Yaskawa INFORM job: OK_R2_O57-69(1)(90,0)OLDMAREK.JBI

/JOB
//NAME OK_R2_O57-69(1)(90,0)OLDMAREK
//POS
///NPOS 679,679,679,19,0,0
///TOOL 0
///POSTYPE PULSE
///PULSE
C00000=-115282,71817,32941,48127,54711,-22306
C00001=-113844,78377,40832,48113,52960,-22533
C00002=-113286,81152,44222,48167,52223,-22657
C00003=-112658,81907,45149,47913,51773,-22558
C00004=-113286,81152,44222,48167,52223,-22657
C00005=-114841,82290,45172,49039,53033,-23084
C00006=-115003,85006,48527,49507,52672,-23414
C00007=-114841,82290,45172,49039,53033,-23084
C00008=-115410,79539,41800,48987,53774,-22957
C00009=-116878,73048,33960,49005,55537,-22725
C00010=-112638,83822,30523,28584,74380,-13794
C00011=-107672,118155,51647,4031,94928,-4029
C00012=-107420,122850,61171,3935,91477,-4062
C00013=-107323,125066,65433,3902,89992,-4078
C00014=-107323,124239,65578,3901,89479,-4094
C00015=-107323,125066,65433,3902,89992,-4078
C00016=-107335,126122,66498,3905,89879,-4086
C00017=-107232,129619,71327,3873,88703,-4090
C00018=-107335,126122,66498,3905,89879,-4086
C00019=-107432,123868,62180,3938,91380,-4069
C00020=-107683,119107,52557,4034,94858,-4034
C00021=-108242,110727,51927,9928,92581,-10453
C00022=-107623,115488,61342,9730,89211,-10523
C00023=-107381,117723,65553,9663,87760,-10558
C00024=-107381,117129,66014,9664,87180,-10602
C00025=-107381,117723,65553,9663,87760,-10558
C00026=-107320,118492,66386,9646,87637,-10548
C00027=-107068,121743,70795,9581,86581,-10547
C00028=-107320,118492,66386,9646,87637,-10548
C00029=-107562,116223,62127,9713,89100,-10512
C00030=-108179,111405,52627,9909,92492,-10440
C00031=-110424,91387,35110,11931,86832,-11135
C00032=-122323,33946,36249,27998,48832,-19209
C00033=-121111,41698,46132,28269,46563,-19325
C00034=-120645,45031,50436,28448,45578,-19411
C00035=-120645,45990,52788,28899,44735,-19701
C00036=-120645,45031,50436,28448,45578,-19411
C00037=-120832,44203,49576,28499,45733,-19457
C00038=-120451,46607,52174,28466,45283,-19410
C00039=-120832,44203,49576,28499,45733,-19457
C00040=-121303,40901,45320,28328,46708,-19376
C00041=-122523,33209,35531,28074,48955,-19270
C00042=-138494,21467,-20962,-13510,88545,-918
C00043=-172308,65494,48979,-45567,35920,22282
C00044=-172307,66906,54819,-48573,33928,23926
C00045=-172639,69838,58273,-49022,33332,24169
C00046=-173239,69159,57471,-48394,33104,23833
C00047=-173424,69192,57512,-48260,33005,23761
C00048=-172268,71224,59921,-49648,33330,24503
C00049=-172150,82507,73646,-52983,31698,26274
C00050=-172069,85080,76852,-53896,31347,26756
C00051=-171567,71541,60313,-50254,33662,24828
C00052=-171245,62238,49417,-48357,35120,23797
C00053=-171365,58220,44512,-47276,35710,23205
C00054=-172568,85923,51709,-38156,42478,18009
C00055=-173210,88622,55081,-38109,41654,18042
C00056=-173399,87523,53708,-37764,41797,17852
C00057=-171913,88923,55458,-39192,42161,18576
C00058=-172373,102262,72497,-41555,39146,20013
C00059=-172364,103826,74533,-41931,38810,20229
C00060=-172120,93439,61160,-39872,41141,19005
C00061=-171772,85324,50969,-38678,42942,18248
C00062=-171214,82198,47055,-38587,43820,18132
C00063=-172412,95660,50695,-34930,47113,15937
C00064=-172941,98291,54078,-34907,46302,16003
C00065=-173393,98042,53756,-34511,46183,15812
C00066=-173582,97646,53244,-34301,46202,15703
C00067=-172217,98411,54230,-35491,46558,16277
C00068=-172267,109740,69033,-37375,43863,17490
C00069=-172235,113172,73586,-38066,43046,17916
C00070=-172202,103053,60251,-36243,45483,16763
C00071=-171971,91033,44794,-34631,48320,15659
C00072=-172583,89506,42865,-33959,48423,15307
C00073=-136545,44574,15947,-43124,46451,20365
C00074=-172050,-124043,-93312,-19428,16171,9287
C00075=-153076,-24082,-53998,12354,68401,18517
C00076=-141616,-19382,-55807,13562,72328,27791
C00077=-136367,-32764,-63918,14399,72043,28923
C00078=-134539,-35777,-64067,14758,71094,29221
C00079=-134539,-36232,-63095,14829,70289,29119
C00080=-134539,-35777,-64067,14758,71094,29221
C00081=-134790,5262,-45049,12672,103577,12599
C00082=-134622,7343,-43237,12633,103510,12643
C00083=-134790,5262,-45049,12672,103577,12599
C00084=-132608,-4947,-51631,7718,96928,11812
C00085=-133594,-4601,-51352,7990,97018,11521
C00086=-132608,-4947,-51631,7718,96928,11812
C00087=-132561,-6063,-53863,7723,97717,11875
C00088=-132436,-8720,-59337,7740,99694,12036
C00089=-132445,-1782,-62924,7952,105415,12403
C00090=-141601,37323,-23290,10329,102010,9516
C00091=-93172,55874,9388,-1843,94357,23900
C00092=-93485,56784,11787,-1769,93341,23816
C00093=-93485,56329,12545,-1767,92641,23826
C00094=-93485,56784,11787,-1769,93341,23816
C00095=-93464,57012,11403,-1775,93695,23818
C00096=-93714,59095,13766,-1718,93307,23745
C00097=-93464,57012,11403,-1775,93695,23818
C00098=-94351,55649,10247,-1575,93690,23540
C00099=-95033,54913,9421,-1421,93808,23324
C00100=-94351,55649,10247,-1575,93690,23540
C00101=-94041,54751,7862,-1648,94701,23624
C00102=-93250,52756,2164,-1838,97197,23834
C00103=-93258,57323,-1415,-1867,101744,23764
C00104=-108708,74058,35602,41753,92549,11625
C00105=-107609,77867,43172,41468,89995,11080
C00106=-107179,79572,46434,41382,88936,10847
C00107=-107179,79487,47575,41378,88368,10623
C00108=-107179,79572,46434,41382,88936,10847
C00109=-85041,17756,-8276,-11251,50625,9461
C00110=-85416,19690,-6470,-10982,50459,9320
C00111=-85041,17756,-8276,-11251,50625,9461
C00112=-87036,75660,30192,-3211,91902,25887
C00113=-87645,74633,28952,-3076,92115,25688
C00114=-87036,75660,30192,-3211,91902,25887
C00115=-86708,74680,27642,-3289,92979,25963
C00116=-85872,72543,21626,-3493,95611,26155
C00117=-85876,74587,19798,-3512,97782,26092
C00118=-86821,26768,-33196,-3418,105774,25582
C00119=-56288,-65443,-100505,-9939,102051,34984
C00120=-94872,-76247,-37251,-15619,10327,-42827
C00121=-113351,-68967,-59155,816,27582,-73246
C00122=-112415,-66495,-57032,-529,27544,-72574
C00123=-112416,-66088,-55565,-540,26850,-72568
C00124=-112415,-66495,-57032,-529,27544,-72574
C00125=-125986,-60936,-52893,34026,33366,-67517
C00126=-125619,-58716,-51713,33325,33568,-67144
C00127=-125986,-60936,-52893,34026,33366,-67517
C00128=-125164,-63316,-53721,33839,32440,-67422
C00129=-123797,-63897,-54019,32563,31806,-66752
C00130=-125164,-63316,-53721,33839,32440,-67422
C00131=-126284,-65474,-55722,34821,32994,-67941
C00132=-120687,-90156,-48971,65843,10407,33929
C00133=-163424,-29173,-12092,69684,68620,47205
C00134=-154639,-8126,3338,68913,63218,49031
C00135=-170775,-70491,-60275,67726,76450,43734
C00136=-168988,-72616,-61292,67687,75067,43782
C00137=-168256,-73449,-61686,67672,74502,43804
C00138=-168255,-73444,-61683,67672,74502,43805
C00139=-168256,-73449,-61686,67672,74502,43804
C00140=-168129,-73592,-61753,67670,74405,43808
C00141=-167340,-74469,-62163,67655,73798,43833
C00142=-168129,-73592,-61753,67670,74405,43808
C00143=-168863,-72760,-61361,67684,74971,43786
C00144=-170655,-70639,-60347,67723,76357,43737
C00145=-172135,-82938,-72310,60788,72518,32969
C00146=-200540,-66438,-67217,63628,100285,-15829
C00147=-127293,-88890,-117674,21964,112183,-47373
C00148=-127884,-113870,-117586,20406,100261,-49782
C00149=-127000,-93154,-82052,19489,96345,-50169
C00150=-123343,-94047,-79271,19637,93420,-49322
C00151=-121848,-94244,-78089,19702,92278,-48969
C00152=-121841,-92834,-76346,19694,91947,-49020
C00153=-121848,-94244,-78089,19702,92278,-48969
C00154=-119969,-93354,-78147,19815,92288,-48290
C00155=-118222,-93288,-78121,19899,91881,-47727
C00156=-119969,-93354,-78147,19815,92288,-48290
C00157=-121462,-93189,-79339,19761,93422,-48643
C00158=-125120,-92380,-82146,19635,96326,-49491
C00159=-116413,-89407,-85315,-11170,94586,69972
C00160=-118284,-91858,-82643,-11111,91478,69605
C00161=-119058,-92674,-81496,-11095,90266,69446
C00162=-119072,-91347,-79783,-11093,89899,69474
C00163=-119058,-92674,-81496,-11095,90266,69446
C00164=-118796,-98042,-83265,-11090,88662,69679
C00165=-118746,-100551,-83769,-11090,87708,69781
C00166=-118796,-98042,-83265,-11090,88662,69679
C00167=-123354,-93602,-81963,-11047,89491,68033
C00168=-125085,-93483,-81915,-11019,89286,67454
C00169=-123354,-93602,-81963,-11047,89491,68033
C00170=-122534,-92869,-83147,-11066,90689,68210
C00171=-120547,-90622,-85912,-11132,93767,68620
C00172=-120571,-90661,-98380,-11386,101275,67925
C00173=-125069,-105236,-119201,46912,96955,7142
C00174=-121279,-99548,-114464,46207,95099,8000
C00175=-119841,-97303,-112552,45921,94382,8319
C00176=-119849,-96483,-111054,45883,94032,8153
C00177=-119841,-97303,-112552,45921,94382,8319
C00178=-121259,-87971,-110760,46601,97668,9229
C00179=-121544,-83907,-109504,46842,98723,9610
C00180=-121259,-87971,-110760,46601,97668,9229
C00181=-122654,-89805,-112582,46929,98462,8982
C00182=-126320,-94321,-117059,47765,100534,8329
C00183=-125132,-111985,-108710,18887,62200,-22139
C00184=-122150,-102499,-103347,17190,63051,-20837
C00185=-121052,-98905,-101202,16573,63333,-20372
C00186=-121051,-97751,-99591,16628,62949,-20429
C00187=-121052,-98905,-101202,16573,63333,-20372
C00188=-120662,-97381,-100799,16308,63770,-20159
C00189=-118912,-97325,-100778,15434,63451,-19540
C00190=-120662,-97381,-100799,16308,63770,-20159
C00191=-120717,-96579,-100674,16290,64103,-20131
C00192=-120723,-93199,-99767,16143,65237,-19969
C00193=-120717,-96579,-100674,16290,64103,-20131
C00194=-121791,-100117,-102825,16885,63842,-20577
C00195=-124704,-109452,-108202,18522,63043,-21827
C00196=-114740,-109793,-107699,-22238,66313,27441
C00197=-118303,-101714,-102676,-20552,66389,26052
C00198=-119630,-98598,-100655,-19919,66404,25543
C00199=-119640,-97443,-99041,-19972,66025,25607
C00200=-119630,-98598,-100655,-19919,66404,25543
C00201=-120869,-98346,-100801,-19339,66320,25087
C00202=-122629,-98310,-100787,-18548,65929,24486
C00203=-120869,-98346,-100801,-19339,66320,25087
C00204=-120753,-95574,-99975,-19267,67213,24978
C00205=-120759,-92226,-99069,-19116,68313,24791
C00206=-120753,-95574,-99975,-19267,67213,24978
C00207=-119475,-98647,-102011,-19875,67204,25461
C00208=-116042,-106621,-107071,-21497,67130,26779
C00209=-113894,-113482,-108593,-25442,60982,30098
C00210=-117729,-104898,-103745,-23262,61171,28471
C00211=-119152,-101582,-101788,-22448,61245,27877
C00212=-119170,-99953,-99618,-22541,60778,27968
C00213=-119152,-101582,-101788,-22448,61245,27877
C00214=-121013,-102333,-103012,-21430,61098,27156
C00215=-123420,-102254,-102982,-20177,60519,26301
C00216=-121013,-102333,-103012,-21430,61098,27156
C00217=-120862,-89775,-98642,-20835,64658,26523
C00218=-120866,-85351,-97357,-20602,66047,26262
C00219=-120862,-89775,-98642,-20835,64658,26523
C00220=-119577,-92842,-100627,-21537,64647,27018
C00221=-116128,-100765,-105545,-23412,64594,28369
C00222=-120616,-96668,-103675,-23957,64374,45643
C00223=-120616,-97077,-101536,-24254,62975,45956
C00224=-120616,-97187,-100661,-24377,62430,46080
C00225=-118869,-97129,-100639,-25236,62958,46664
C00226=-120614,-98300,-102259,-24293,62807,45995
C00227=-120617,-94441,-109322,-23464,92098,42048
C00228=-120616,-97113,-101199,-23421,86229,43199
C00229=-120616,-97196,-100378,-23430,85724,43299
C00230=-120616,-97068,-101477,-23418,86408,43164
C00231=-120616,-96536,-104145,-23405,88172,42819
C00232=-120615,-97089,-97846,-24331,46439,48575
C00233=-120614,-96205,-89198,-26458,42021,49913
C00234=-120613,-95813,-87227,-26966,41113,50220
C00235=-120613,-95637,-86431,-27175,40755,50344
C00236=-118868,-95589,-86413,-28580,41350,51125
C00237=-120611,-96965,-88121,-26990,41076,50233
C00238=-120617,-95981,-105264,-23408,89069,42643
C00239=-120616,-96766,-101896,-23413,86788,43090
C00240=-120616,-96795,-102141,-18817,118956,36582
C00241=-120616,-96568,-103294,-18987,119739,36439
C00242=-120617,-95735,-106079,-19458,121767,36056
C00243=-120683,-72727,-118704,-1403,106780,1205
C00244=-120616,-97110,-101484,23732,56591,-46685
C00245=-120615,-97329,-97421,24453,54195,-47265
C00246=-120615,-97216,-95276,24833,53043,-47558
C00247=-120615,-97137,-94405,24989,52592,-47675
C00248=-120613,-98372,-96050,24869,52935,-47585
C00249=-122362,-97116,-94396,26052,53130,-48332
C00250=-120617,-95602,-107135,23341,90098,-42167
C00251=-120617,-96025,-106062,23332,89289,-42325
C00252=-120617,-96280,-105304,23328,88738,-42432
C00253=-120617,-95942,-106325,23333,89477,-42288
C00254=-120617,-94838,-108784,23367,91395,-41914
C00255=-120619,-89077,-114974,23678,97628,-40680
C00256=-119375,-87803,-114046,-9627,73434,-76892
C00257=-119874,-91001,-111320,-9540,70103,-76790
C00258=-120074,-92022,-110137,-9508,68845,-76756
C00259=-120388,-88035,-108953,-9268,70114,-76963
C00260=-120068,-92699,-111595,-9479,69387,-76797
C00261=-120617,-92323,-109789,-9348,67950,-76861
C00262=-120617,-92636,-109412,-9435,67087,-76774
C00263=-120617,-92966,-108935,-9385,65680,-76698
C00264=-120617,-93485,-108112,-8702,63167,-76584
C00265=-120617,-93807,-107566,-7310,61334,-76551
C00266=-120617,-93899,-107425,-5913,60596,-76588
C00267=-120617,-91887,-110532,-5160,63404,-76609
C00268=-120617,-91830,-110616,-4244,63440,-76636
C00269=-120617,-91600,-110911,-2665,64017,-76695
C00270=-120618,-91126,-111456,-1065,65432,-76762
C00271=-120618,-90436,-112164,126,67515,-76814
C00272=-120618,-89799,-112749,669,69377,-76843
C00273=-120618,-88579,-113586,734,71430,-76721
C00274=-120618,-87737,-114188,674,73665,-76767
C00275=-120618,-86710,-114840,-40,76341,-76871
C00276=-120619,-85981,-115253,-1370,78289,-77032
C00277=-120619,-85769,-115356,-2649,79041,-77176
C00278=-118258,-89310,-112812,-4565,75923,-76275
C00279=-117029,-89279,-112689,-5985,75998,-75947
C00280=-115084,-89307,-112300,-8369,75681,-75412
C00281=-113300,-89514,-111627,-10775,74614,-74872
C00282=-112191,-89952,-110802,-12600,72842,-74453
C00283=-112162,-90329,-110382,-13115,71673,-74372
C00284=-116808,-91534,-110372,-11031,70029,-75758
C00285=-120074,-92022,-110137,-9508,68845,-76756
C00286=-119874,-91001,-111320,-9540,70103,-76790
C00287=-119375,-87803,-114046,-9627,73434,-76892
C00288=-120613,-96141,-86612,-20456,81391,53018
C00289=-120613,-95201,-83022,-20541,79769,53295
C00290=-120613,-94772,-81561,-20579,79132,53405
C00291=-119108,-93506,-81277,-20755,79958,53812
C00292=-120703,-96226,-83293,-20548,79408,53324
C00293=-120613,-95341,-83418,-16256,85806,57019
C00294=-120612,-93770,-78536,-16295,83694,57299
C00295=-120612,-93943,-79000,-13291,89893,68155
C00296=-120613,-94474,-80645,-13297,90613,68078
C00297=-120613,-95649,-84682,-13324,92446,67881
C00298=-120615,-97441,-93706,-13451,96957,67391
C00299=-117944,-114132,-91182,23549,57658,-33742
C00300=-120612,-94052,-79174,30375,49115,-27391
C00301=-120612,-92306,-74262,31338,47277,-28046
C00302=-120611,-91624,-72518,31687,46656,-28277
C00303=-120611,-91343,-71816,31829,46409,-28371
C00304=-120609,-92783,-73582,31657,46706,-28257
C00305=-122365,-91326,-71808,32798,47083,-29054
C00306=-120614,-96423,-87542,23693,78601,-44429
C00307=-120612,-92192,-73989,24270,72943,-45595
C00308=-120612,-92493,-74805,23528,86971,-60762
C00309=-120612,-93040,-76284,23523,87550,-60648
C00310=-120612,-94304,-79928,23524,89017,-60360
C00311=-192979,-49879,-84133,31949,90821,-59300
C00312=-226136,-49296,-77583,43048,96139,-60221
C00313=-194231,-43574,-37464,64429,96533,35524
C00314=-168190,-921,2356,69742,86936,65420
C00315=-157686,-14873,-8721,69811,79682,66593
C00316=-155170,-17431,-10634,69793,77924,66853
C00317=-154140,-18406,-11354,69782,77205,66960
C00318=-154960,-19735,-12328,69815,77730,66818
C00319=-154139,-18877,-12975,69638,77486,67291
C00320=-152416,-19959,-12491,68149,70274,62953
C00321=-151462,-20771,-13080,67326,65877,57651
C00322=-150584,-21490,-13598,66880,61935,51327
C00323=-149448,-22378,-14235,66195,57985,45258
C00324=-150364,-21665,-13724,66599,59939,44567
C00325=-146294,-24621,-15825,64622,49633,44461
C00326=-147024,-24129,-15478,65026,50858,44122
C00327=-148183,-23314,-14902,65711,53127,43519
C00328=-150746,-21357,-13503,66515,56405,42739
C00329=-151844,-20450,-12847,67017,58691,42205
C00330=-154160,-18394,-11345,67568,61790,41547
C00331=-155150,-17454,-10651,67918,63984,41080
C00332=-156307,-16307,-9798,68285,66690,40524
C00333=-158578,-13896,-7981,68632,70174,39857
C00334=-158236,-14274,-8267,68563,69306,40027
C00335=-158768,-13688,-7823,68593,69674,39964
C00336=-160083,-12191,-6676,68663,70584,39811
C00337=-163356,-38025,-17867,70039,68206,46757
C00338=-171321,-47804,-23743,70196,73038,45095
C00339=-120855,-117042,-83065,287,50429,-281
C00340=-120852,-56541,-79529,233,79340,-219
C00341=-120696,51333,26745,175,69370,-180
C00342=-120686,107948,75662,172,68359,-178
C00343=-120686,108277,78684,174,66668,-180
C00344=-120686,108491,80003,175,65967,-181
C00345=-120685,108330,78544,174,66782,-180
C00346=-120704,104314,74519,181,67195,-186
C00347=-120686,108513,80202,3786,65964,-3429
C00348=-120686,108564,80691,8354,65806,-7433
C00349=-120686,108545,80707,11489,66690,-7514
C00350=-120686,108555,80692,12508,67155,-8479
C00351=-120686,108564,80762,15450,68398,-11287
C00352=-120686,108549,80793,17539,69495,-16102
C00353=-120686,109188,83963,29512,74271,-26746
C00354=-120686,108838,82574,29428,74862,-26590
C00355=-120686,108172,79385,29242,76284,-26220
C00356=-120686,107962,76375,6322,66410,-5366
C00357=-120686,108346,79348,6400,64788,-5455
C00358=-120686,108578,80641,6435,64115,-5493
C00359=-120686,108293,79018,6392,64962,-5445
C00360=-120992,104893,75799,6510,65219,-5544
C00361=-120686,108263,79465,19749,71998,-15740
C00362=-120686,108289,79502,19750,71989,-15741
C00363=-120686,109192,84126,33583,78410,-30786
C00364=-120686,108845,82779,33520,78957,-30620
C00365=-120686,108177,79678,33383,80274,-30223
C00366=-146832,94827,54018,-31343,96631,42054
C00367=-156862,88199,54516,-55770,96758,71489
C00368=-156858,88352,61458,-55305,94312,73083
C00369=-157852,91445,67330,-55099,92539,73648
C00370=-158245,92835,69884,-55033,91801,73892
C00371=-157951,96204,74186,-54996,91433,74294
C00372=-157784,91273,67188,-55102,92578,73662
C00373=-158040,92399,69988,-55026,91755,74041
C00374=-159291,95627,71523,-51291,93332,81554
C00375=-160209,98279,73182,-48482,94322,83905
C00376=-159956,97162,70645,-48575,95125,83623
C00377=-159321,94794,64867,-48849,97041,82959
C00378=-174197,80542,71118,-15802,102714,62389
C00379=-174195,80556,71135,-15802,102711,62390
C00380=-174195,80561,71142,-15801,102710,62390
C00381=-173773,83477,74756,-15654,102092,62625
C00382=-174194,79765,68888,-15876,103653,62265
C00383=-174199,80535,71109,-11568,105990,64366
C00384=-174198,80539,71114,-12074,105866,67869
C00385=-174201,80518,71089,-8660,108894,72599
C00386=-174202,80510,71078,-8661,108896,72599
C00387=-174205,80488,71052,-8662,108901,72597
C00388=-174210,80448,71002,-8664,108910,72595
C00389=-160796,99181,68474,-21491,79626,-54117
C00390=-160795,99200,68498,-21491,79622,-54116
C00391=-160795,99207,68507,-21491,79620,-54116
C00392=-160747,98987,66984,-21457,80402,-54239
C00393=-161332,101028,70752,-21395,79065,-54211
C00394=-160795,99207,68507,-21491,79620,-54116
C00395=-160795,99200,68498,-21491,79622,-54116
C00396=-160796,99181,68474,-21491,79626,-54117
C00397=-156887,88424,61529,-55303,94292,73080
C00398=-157880,91522,67408,-55097,92517,73646
C00399=-158273,92915,69967,-55032,91779,73890
C00400=-157979,96289,74274,-54994,91410,74293
C00401=-157812,91350,67266,-55100,92556,73660
C00402=-158068,92478,70069,-55024,91733,74039
C00403=-159318,95712,71612,-51289,93309,81552
C00404=-160236,98368,73278,-48480,94299,83903
C00405=-159983,97249,70737,-48574,95102,83621
C00406=-159349,94875,64951,-48847,97020,82956
C00407=-174197,80542,71118,-15802,102714,62389
C00408=-174195,80555,71135,-15802,102711,62390
C00409=-174195,80561,71141,-15801,102710,62390
C00410=-173773,83477,74755,-15654,102093,62624
C00411=-174194,79764,68887,-15876,103653,62265
C00412=-174199,80534,71109,-11568,105990,64366
C00413=-174198,80538,71114,-12074,105866,67869
C00414=-174201,80518,71088,-8660,108894,72599
C00415=-174202,80509,71078,-8661,108896,72599
C00416=-174205,80488,71051,-8662,108901,72597
C00417=-174210,80448,71002,-8664,108910,72595
C00418=-160796,99181,68473,-21491,79626,-54117
C00419=-160795,99199,68497,-21491,79622,-54116
C00420=-160795,99206,68506,-21491,79620,-54116
C00421=-160747,98986,66983,-21457,80402,-54239
C00422=-161332,101028,70752,-21395,79065,-54211
C00423=-160795,99206,68506,-21491,79620,-54116
C00424=-160795,99199,68497,-21491,79622,-54116
C00425=-160796,99181,68473,-21491,79626,-54117
C00426=-156915,88496,61599,-55301,94271,73077
C00427=-157907,91600,67487,-55096,92496,73644
C00428=-158301,92995,70050,-55030,91757,73888
C00429=-158006,96373,74363,-54993,91387,74291
C00430=-157840,91427,67345,-55098,92535,73658
C00431=-158096,92558,70151,-55023,91711,74037
C00432=-159346,95797,71702,-51288,93287,81550
C00433=-160263,98458,73375,-48479,94275,83902
C00434=-160010,97336,70829,-48572,95080,83619
C00435=-159376,94956,65035,-48845,96998,82954
C00436=-174177,99010,68236,-17004,113547,60859
C00437=-174175,99024,68253,-17003,113544,60860
C00438=-174175,99029,68260,-17002,113542,60860
C00439=-173779,101892,71964,-16797,112849,61119
C00440=-174174,98966,66934,-17118,114293,60744
C00441=-174178,99003,68226,-12626,117020,63205
C00442=-174178,99007,68232,-13170,116875,66659
C00443=-174181,98987,68205,-9575,120026,71701
C00444=-174182,98978,68194,-9576,120028,71701
C00445=-174185,98957,68167,-9578,120033,71699
C00446=-174189,98918,68117,-9580,120044,71697
C00447=-160796,99180,68472,-21491,79627,-54117
C00448=-160795,99198,68496,-21491,79622,-54116
C00449=-160795,99206,68506,-21491,79620,-54116
C00450=-160747,98986,66982,-21457,80402,-54239
C00451=-161332,101027,70751,-21395,79065,-54211
C00452=-160795,99206,68506,-21491,79620,-54116
C00453=-160795,99198,68496,-21491,79622,-54116
C00454=-160796,99180,68472,-21491,79627,-54117
C00455=-160394,63694,17038,-3651,83782,-73608
C00456=-190015,-23229,-64935,6709,90053,81130
C00457=-200263,9721,-38620,10181,91724,78169
C00458=-174135,-51322,-31088,61328,33879,50976
C00459=-174134,-51319,-31087,61327,33879,50977
C00460=-174133,-51978,-32760,60430,34229,51462
C00461=-175008,-52913,-31974,62066,34294,50529
C00462=-174165,-51376,-31119,68078,48326,49661
C00463=-174167,-51380,-31120,67173,48568,55955
C00464=-174192,-51426,-31146,69828,61157,64510
C00465=-174196,-51432,-31150,69829,61158,64509
C00466=-160788,-42263,-32458,15580,47921,8219
C00467=-160788,-42263,-32458,15580,47921,8219
C00468=-159909,-43388,-33874,14966,48039,8647
C00469=-161405,-44119,-33586,16024,47791,7908
C00470=-160787,-42259,-32456,15583,47920,8217
C00471=-160784,-42250,-32450,15581,47921,8219
C00472=-160783,-42246,-32448,15576,47922,8221
C00473=-160783,-42246,-32448,15576,47922,8221
C00474=-146637,-39575,-34461,6046,48590,14746
C00475=-174196,-30579,-7118,69980,41906,48750
C00476=-174191,-30568,-7111,69979,41904,48752
C00477=-174188,-30559,-7105,69977,41901,48753
C00478=-174186,-30555,-7102,69976,41901,48754
C00479=-174186,-31355,-8970,69207,42176,49221
C00480=-174962,-32094,-8117,70258,42357,48510
C00481=-174194,-30569,-7112,71825,47591,46341
C00482=-174196,-30575,-7115,70727,48120,54586
C00483=-174217,-30615,-7142,71977,59732,62495
C00484=-174219,-30621,-7146,71977,59734,62495
C00485=-174226,-30637,-7157,71978,59738,62493
C00486=-174235,-30659,-7171,71979,59742,62491
C00487=-160826,40415,13631,53464,67015,37205
C00488=-160826,40346,14725,53699,66583,36924
C00489=-160826,40419,13556,53448,67045,37224
C00490=-161205,38368,12671,53745,66948,36941
C00491=-160829,40326,14814,56358,71294,34357
C00492=-160833,40301,19018,62693,68392,39666
C00493=-160845,41308,28286,76228,74003,43895
C00494=-160845,41098,27088,76066,74172,44186
C00495=-160847,40669,24199,75673,74598,44902
C00496=-160844,40222,15431,74465,76073,47261
C00497=-107800,-52207,-58944,57218,40703,55200
C00498=-68476,-97884,-84022,-50002,23247,45036
C00499=-66040,-99229,-83751,-49838,32871,-40371
C00500=-120096,-126434,-88762,51835,16555,74218
C00501=-135002,-84086,-73993,57476,43061,70498
C00502=-132040,-84680,-73570,56549,40955,71010
C00503=-130846,-84617,-72526,56532,39890,71007
C00504=-131406,-87072,-73560,57444,39877,70476
C00505=-130845,-85029,-73961,55869,40275,71397
C00506=-120674,-85352,-72158,6203,19725,75700
C00507=-120674,-85360,-72169,6198,19735,75701
C00508=-120674,-85375,-72170,13051,20123,72466
C00509=-120675,-85403,-72185,17568,20556,70326
C00510=-120675,-85415,-72191,21840,21109,68297
C00511=-120675,-85426,-72197,23876,21425,67327
C00512=-120675,-85665,-72942,26166,23375,58358
C00513=-120894,-85673,-72945,29533,24131,56524
C00514=-120675,-85602,-72710,24864,23359,52833
C00515=-120675,-85601,-72708,24818,23350,52837
C00516=-120675,-85948,-73873,24306,23842,53086
C00517=-120674,-86249,-74914,23862,24287,53303
C00518=-120096,-126434,-88762,51835,16555,74218
C00519=-66040,-99229,-83751,-49838,32871,-40371
C00520=-124550,-62434,-86348,-29573,82344,852
C00521=-123235,4833,-40404,-29868,88268,-211
C00522=-160797,40338,30634,-17216,54639,-7315
C00523=-160798,40335,30631,-17216,54639,-7316
C00524=-160798,40334,30630,-17216,54639,-7316
C00525=-160254,39145,28669,-17377,55324,-7200
C00526=-161179,38217,28428,-16962,54815,-7509
C00527=-160797,40338,30635,-17214,54636,-7317
C00528=-160796,40349,30645,-17215,54635,-7316
C00529=-160795,40353,30650,-17218,54637,-7314
C00530=-160795,40355,30652,-17218,54637,-7314
C00531=-160794,40358,30655,-17219,54637,-7314
C00532=-134055,6389,-12297,-27269,70214,305
C00533=-134055,6386,-12300,-27269,70214,304
C00534=-134056,6385,-12301,-27269,70214,304
C00535=-133336,6111,-13253,-27465,70843,431
C00536=-134209,4258,-14137,-27207,70198,248
C00537=-134055,6389,-12297,-27268,70211,304
C00538=-134055,6399,-12288,-27268,70211,304
C00539=-134055,6404,-12285,-27269,70214,305
C00540=-134054,6405,-12283,-27269,70214,305
C00541=-134054,6409,-12280,-27270,70214,305
C00542=-134054,6381,-12304,-27269,70214,305
C00543=-107307,118486,66692,6711,86217,-7198
C00544=-107308,118513,66728,6711,86209,-7198
C00545=-107308,118524,66743,6711,86205,-7199
C00546=-107412,115203,62263,6738,87257,-7176
C00547=-107308,119140,66313,6709,86782,-7168
C00548=-107310,118572,66809,-801,85169,-3247
C00549=-107308,118507,66720,-802,85190,-3246
C00550=-107307,118486,66692,-801,85189,-3246
C00551=-107307,118478,66681,-801,85191,-3246
C00552=-107306,118457,66653,-801,85198,-3245
C00553=-107310,127854,66507,14056,94097,-10874
C00554=-107310,125830,66726,14028,92956,-11004
C00555=-107310,125066,66876,14018,92485,-11057
C00556=-107310,125885,66724,14029,92985,-11000
C00557=-107565,122036,62719,14104,93498,-11023
C00558=-107311,125084,66901,14017,92482,-11058
C00559=-107312,125131,66974,14017,92463,-11061
C00560=-107313,125147,66999,14019,92452,-11062
C00561=-107313,125910,66849,14028,92923,-11008
C00562=-107313,127932,66629,14055,94064,-10878
C00563=-132655,20555,-34602,20500,105579,-17250
C00564=-120395,-75677,-109491,17431,99945,-14261
C00565=-120731,-81008,-115648,-105,86416,-81801
C00566=-120675,-24649,-47159,-132,73228,-81771
C00567=-120676,-24635,-47149,-131,73230,-81771
C00568=-120677,-24629,-47145,-131,73230,-81771
C00569=-120676,-24365,-48211,-131,74022,-81772
C00570=-121750,-24621,-47139,317,73232,-82133
C00571=-120677,-24629,-47145,-131,73230,-81771
C00572=-120676,-24635,-47149,-131,73230,-81771
C00573=-120675,-24649,-47159,-132,73228,-81771
C00574=-86683,-40445,-63075,-13763,77736,-70672
C00575=-103499,26970,-9106,-7161,77072,-76192
C00576=-140778,108087,66612,-20508,92087,-48724
C00577=-140778,108110,66641,-20508,92080,-48723
C00578=-140777,108132,66670,-20508,92074,-48722
C00579=-140777,108059,66946,-20503,91880,-48688
C00580=-140777,108336,66063,-20521,92524,-48798
C00581=-141368,108983,68165,-20410,91478,-48827
C00582=-140777,108060,66945,-20503,91881,-48689
C00583=-140777,108132,66670,-20508,92074,-48722
C00584=-140778,108110,66641,-20508,92080,-48723
C00585=-140778,108110,66641,-20508,92080,-48723
C00586=-140777,108131,66669,-20508,92074,-48722
C00587=-140777,108063,66930,-20504,91891,-48690
C00588=-140777,108340,66048,-20521,92535,-48800
C00589=-141368,108987,68148,-20410,91489,-48829
C00590=-140777,108063,66929,-20504,91892,-48691
C00591=-140777,108131,66669,-20508,92075,-48722
C00592=-140778,108109,66640,-20508,92081,-48723
C00593=-140778,108086,66610,-20508,92087,-48724
C00594=-125618,13255,-41495,-24522,112345,-47401
C00595=-160865,108111,66627,-28476,101259,-43958
C00596=-160864,108058,66881,-28455,101097,-43917
C00597=-160864,107744,68124,-28354,100277,-43712
C00598=-160867,111482,73064,-28240,99285,-43467
C00599=-160864,107969,67173,-28430,100897,-43867
C00600=-160866,107730,68106,-28354,100280,-43713
C00601=-160865,108044,66863,-28456,101100,-43918
C00602=-160866,108097,66609,-28477,101262,-43960
C00603=-160868,107404,70021,-43698,97330,-44642
C00604=-160870,107239,73702,-43453,95599,-43897
C00605=-160870,107318,75365,-43366,94873,-43587
C00606=-160873,111572,80985,-43267,93932,-43187
C00607=-160870,107239,74018,-43435,95456,-43836
C00608=-160872,107302,75345,-43366,94876,-43589
C00609=-160871,107223,73682,-43453,95602,-43899
C00610=-160869,107389,70003,-43699,97332,-44644
C00611=-160874,107343,69924,-43701,97348,-44653
C00612=-160876,107172,73597,-43455,95618,-43908
C00613=-160876,107248,75256,-43368,94893,-43598
C00614=-160879,111493,80863,-43269,93954,-43200
C00615=-160876,107172,73912,-43437,95475,-43847
C00616=-160878,107233,75236,-43368,94896,-43600
C00617=-160877,107157,73577,-43456,95621,-43910
C00618=-160875,107329,69906,-43702,97350,-44654
C00619=-160864,108120,66638,-19225,80465,79642
C00620=-160865,107719,68195,-19283,79364,79817
C00621=-160866,107492,69457,-19333,78518,79953
C00622=-160869,111315,74506,-19404,77437,80127
C00623=-160866,107660,68433,-19293,79196,79844
C00624=-160867,107478,69438,-19333,78522,79952
C00625=-160867,107705,68176,-19283,79367,79816
C00626=-160866,108106,66620,-19225,80469,79640
C00627=-132676,28155,-16568,-22865,92034,69453
C00628=-92317,-113799,-85959,-30812,71744,72455
C00629=-96628,-112770,-82257,-30552,68664,71557
C00630=-98379,-112217,-80723,-30431,67461,71175
C00631=-98379,-113112,-82315,-30328,67913,71047
C00632=-96411,-111626,-80828,-30637,68489,71696
C00633=-99549,-107096,-79063,-29940,68444,70416
C00634=-110919,-6166,-22977,-25496,80141,63102
C00635=-111160,-1881,-19489,-25434,80119,63017
C00636=-110380,-1847,-20752,-25579,81075,63097
C00637=-108430,-1542,-23732,-25960,83467,63288
C00638=-108435,-915,-27375,-25886,85783,62776
C00639=-136677,-6918,-22174,6754,67616,76224
C00640=-136566,-5518,-16965,6830,65137,76119
C00641=-136522,-4871,-14806,6865,64144,76076
C00642=-136522,-4996,-16154,6823,64904,76122
C00643=-137450,-4424,-14445,7266,64232,75736
C00644=-136149,-648,-11341,6701,64150,76216
C00645=-132512,59658,48248,5392,58225,77290
C00646=-132303,65388,54850,5360,57097,77317
C00647=-132326,64033,51617,5297,58386,77372
C00648=-132385,61171,44202,5165,61470,77495
C00649=-132391,60136,34710,4949,66760,77726
C00650=-143497,-18954,-38514,21083,45207,71474
C00651=-176671,-139811,-87877,67758,38624,43913
C00652=-136240,-146222,-94929,40423,15519,61887
C00653=-125315,3993,-19530,4296,42519,79792
C00654=-145240,-23853,-59157,-64862,65259,25544
C00655=-174199,98804,67970,-56398,33452,34356
C00656=-174204,98773,67929,-56383,33454,34349
C00657=-174205,98760,67913,-56378,33455,34346
C00658=-173589,98179,67166,-56638,33912,34445
C00659=-174310,95327,63510,-55123,33943,33677
C00660=-174204,98772,67928,-56383,33454,34348
C00661=-174188,123224,126678,-97713,27011,55419
C00662=-174191,99984,75379,-23783,43000,33177
C00663=-174189,99848,74689,-23634,43326,33085
C00664=-174185,99559,73033,-23279,44129,32863
C00665=-157452,-25092,-21559,-39199,52444,33566
C00666=-125692,-17579,-45729,-6567,64267,14209
C00667=-120682,108614,67309,63483,51839,-27699
C00668=-120682,108638,67340,63488,51836,-27703
C00669=-120682,108647,67352,63490,51834,-27704
C00670=-120457,105438,63131,62730,52144,-27175
C00671=-121241,110102,69274,64045,51982,-28035
C00672=-120682,108660,67370,63493,51832,-27706
C00673=-120686,108807,67564,63525,51814,-27729
C00674=-120686,108821,67582,63528,51813,-27732
C00675=-120686,108811,67569,63526,51814,-27730
C00676=-120686,108788,67539,63521,51817,-27727
C00677=-142392,7744,-2374,75487,63080,-35362
C00678=-109819,-108660,-86263,20744,34640,-7165
BC00000=315867,805754,283188
BC00001=315867,805754,283188
BC00002=315867,805754,283188
BC00003=315867,805754,283188
BC00004=315867,805754,283188
BC00005=315867,805754,283188
BC00006=315867,805754,283188
BC00007=315867,805754,283188
BC00008=315867,805754,283188
BC00009=315867,805754,283188
BC00010=307549,815674,160012
BC00011=296747,828556,53
BC00012=296747,828556,53
BC00013=296747,828556,53
BC00014=296747,828556,53
BC00015=296747,828556,53
BC00016=296747,828556,53
BC00017=296747,828556,53
BC00018=296747,828556,53
BC00019=296747,828556,53
BC00020=296747,828556,53
BC00021=306135,825328,64240
BC00022=306135,825328,64240
BC00023=306135,825328,64240
BC00024=306135,825328,64240
BC00025=306135,825328,64240
BC00026=306135,825328,64240
BC00027=306135,825328,64240
BC00028=306135,825328,64240
BC00029=306135,825328,64240
BC00030=306135,825328,64240
BC00031=299623,822444,97950
BC00032=269464,809087,254083
BC00033=269464,809087,254083
BC00034=269464,809087,254083
BC00035=269464,809087,254083
BC00036=269464,809087,254083
BC00037=269464,809087,254083
BC00038=269464,809087,254083
BC00039=269464,809087,254083
BC00040=269464,809087,254083
BC00041=269464,809087,254083
BC00042=302810,780106,176804
BC00043=352775,839220,64861
BC00044=352775,839220,64861
BC00045=352775,839220,64861
BC00046=352775,839220,64861
BC00047=352775,839220,64858
BC00048=352775,839220,64861
BC00049=352775,839220,64861
BC00050=352775,839220,64861
BC00051=352775,839220,64861
BC00052=352775,839220,64861
BC00053=352775,839220,64861
BC00054=364144,825211,174172
BC00055=364144,825211,174172
BC00056=364144,825211,174172
BC00057=364144,825211,174172
BC00058=364144,825211,174172
BC00059=364144,825211,174172
BC00060=364144,825211,174172
BC00061=364144,825211,174172
BC00062=364144,825211,174172
BC00063=368581,821126,335712
BC00064=368581,821126,335712
BC00065=368581,821126,335712
BC00066=368581,821126,335712
BC00067=368581,821126,335712
BC00068=368581,821126,335712
BC00069=368581,821126,335712
BC00070=368581,821126,335712
BC00071=368581,821126,335712
BC00072=368581,821126,335712
BC00073=348377,717029,399871
BC00074=348377,717029,399871
BC00075=259018,665141,117968
BC00076=222101,690544,21502
BC00077=213912,696059,562
BC00078=213892,696192,53
BC00079=213892,696192,53
BC00080=213892,696192,53
BC00081=213892,696192,53
BC00082=213892,696192,53
BC00083=213892,696192,53
BC00084=213892,696192,53
BC00085=213892,696192,53
BC00086=213892,696192,53
BC00087=213892,696192,53
BC00088=213892,696192,53
BC00089=213892,696192,53
BC00090=227277,681725,16932
BC00091=99554,684314,33740
BC00092=99554,684314,33740
BC00093=99554,684314,33740
BC00094=99554,684314,33740
BC00095=99554,684314,33740
BC00096=99554,684314,33740
BC00097=99554,684314,33740
BC00098=99554,684314,33740
BC00099=99554,684314,33740
BC00100=99554,684314,33740
BC00101=99554,684314,33740
BC00102=99554,684314,33740
BC00103=99554,684314,33740
BC00104=69020,711056,11217
BC00105=69020,711056,11217
BC00106=69020,711056,11217
BC00107=69020,711056,11217
BC00108=69020,711056,11217
BC00109=69020,711056,11217
BC00110=69020,711056,11217
BC00111=69020,711056,11217
BC00112=69020,711056,11217
BC00113=69020,711056,11217
BC00114=69020,711056,11217
BC00115=69020,711056,11217
BC00116=69020,711056,11217
BC00117=69020,711056,11217
BC00118=69020,711056,11217
BC00119=69020,711056,11217
BC00120=224,677200,247480
BC00121=7166,683025,94113
BC00122=7166,683025,94113
BC00123=7166,683025,94113
BC00124=7166,683025,94113
BC00125=7166,683025,94113
BC00126=7166,683025,94113
BC00127=7166,683025,94113
BC00128=7166,683025,94113
BC00129=7166,683025,94113
BC00130=7166,683025,94113
BC00131=7166,683025,94113
BC00132=1273,683756,232707
BC00133=15,671225,229408
BC00134=15,671225,229408
BC00135=15,740768,89927
BC00136=15,744982,70925
BC00137=15,746667,63325
BC00138=15,746669,55259
BC00139=15,746667,63325
BC00140=15,747562,63916
BC00141=15,749347,63919
BC00142=15,747562,63916
BC00143=15,745877,71517
BC00144=15,741663,90519
BC00145=4579,733665,218396
BC00146=80822,696048,563603
BC00147=35157,680076,1075175
BC00148=35157,770360,1075175
BC00149=35157,771590,1075175
BC00150=35157,771590,1075175
BC00151=35157,771590,1075175
BC00152=35157,771590,1075175
BC00153=35157,771590,1075175
BC00154=35157,771590,1075175
BC00155=35157,771590,1075175
BC00156=35157,771590,1075175
BC00157=35157,771590,1075175
BC00158=35157,771590,1075175
BC00159=42268,766384,1075175
BC00160=42268,766384,1075175
BC00161=42268,766384,1075175
BC00162=42268,766384,1075175
BC00163=42268,766384,1075175
BC00164=42268,766384,1075175
BC00165=42268,766384,1075175
BC00166=42268,766384,1075175
BC00167=42268,766384,1075175
BC00168=42268,766384,1075175
BC00169=42268,766384,1075175
BC00170=42268,766384,1075175
BC00171=42268,766384,1075175
BC00172=42268,766384,1075175
BC00173=298709,942704,1075175
BC00174=298709,942704,1075175
BC00175=298709,942704,1075175
BC00176=298709,942704,1075175
BC00177=298709,942704,1075175
BC00178=298709,942704,1075175
BC00179=298709,942704,1075175
BC00180=298709,942704,1075175
BC00181=298709,942704,1075175
BC00182=298709,942704,1075175
BC00183=146550,860437,1075175
BC00184=146550,860437,1075175
BC00185=146550,860437,1075175
BC00186=146550,860437,1075175
BC00187=146550,860437,1075175
BC00188=146550,860437,1075175
BC00189=146550,860437,1075175
BC00190=146550,860437,1075175
BC00191=146550,860437,1075175
BC00192=146550,860437,1075175
BC00193=146550,860437,1075175
BC00194=146550,860437,1075175
BC00195=146550,860437,1075175
BC00196=175516,858216,1075175
BC00197=175516,858216,1075175
BC00198=175516,858216,1075175
BC00199=175516,858216,1075175
BC00200=175516,858216,1075175
BC00201=175516,858216,1075175
BC00202=175516,858216,1075175
BC00203=175516,858216,1075175
BC00204=175516,858216,1075175
BC00205=175516,858216,1075175
BC00206=175516,858216,1075175
BC00207=175516,858216,1075175
BC00208=175516,858216,1075175
BC00209=129379,842262,1075175
BC00210=129379,842262,1075175
BC00211=129379,842262,1075175
BC00212=129379,842262,1075175
BC00213=129379,842262,1075175
BC00214=129379,842262,1075175
BC00215=129379,842262,1075175
BC00216=129379,842262,1075175
BC00217=129379,842262,1075175
BC00218=129379,842262,1075175
BC00219=129379,842262,1075175
BC00220=129379,842262,1075175
BC00221=129379,842262,1075175
BC00222=139961,848993,1075175
BC00223=134509,852639,1075175
BC00224=132328,854097,1075175
BC00225=132328,854097,1075175
BC00226=132328,854097,1075175
BC00227=135319,889592,1075175
BC00228=135515,843339,1075175
BC00229=135533,839010,1075175
BC00230=137778,838528,1075175
BC00231=143390,837322,1075175
BC00232=181476,833990,1075175
BC00233=181497,833993,1075175
BC00234=176461,838909,1075175
BC00235=174447,840875,1075175
BC00236=174447,840875,1075175
BC00237=174447,840875,1075175
BC00238=184682,893133,1075175
BC00239=184761,874546,1075175
BC00240=171695,925810,1075175
BC00241=173642,926615,1075175
BC00242=178507,928628,1075175
BC00243=157894,860706,1075175
BC00244=129351,852868,1075175
BC00245=129362,852869,1075175
BC00246=134638,857107,1075175
BC00247=136749,858802,1075175
BC00248=136749,858802,1075175
BC00249=136749,858802,1075175
BC00250=130870,903314,1075175
BC00251=130896,897077,1075175
BC00252=130915,892748,1075175
BC00253=128672,892249,1075175
BC00254=123064,891002,1075175
BC00255=123043,890999,1075175
BC00256=398174,868421,1075175
BC00257=398174,870933,1075175
BC00258=398174,871937,1075175
BC00259=398174,871937,1075175
BC00260=398174,871937,1075175
BC00261=394352,870441,1075175
BC00262=388592,868759,1075175
BC00263=387589,867306,1075175
BC00264=385371,864886,1075175
BC00265=382181,863315,1075175
BC00266=379391,863000,1075175
BC00267=374333,882550,1075175
BC00268=372644,882866,1075175
BC00269=369951,883814,1075175
BC00270=367426,885531,1075175
BC00271=365771,887828,1075175
BC00272=365391,889807,1075175
BC00273=387166,894783,1075175
BC00274=388029,896988,1075175
BC00275=390107,899473,1075175
BC00276=393233,901117,1075175
BC00277=396017,901463,1075175
BC00278=398174,881975,1075175
BC00279=398174,881649,1075175
BC00280=398174,880650,1075175
BC00281=398174,878842,1075175
BC00282=398174,876454,1075175
BC00283=398174,875055,1075175
BC00284=398174,873339,1075175
BC00285=398174,871937,1075175
BC00286=398174,870933,1075175
BC00287=398174,868421,1075175
BC00288=48419,769941,1075175
BC00289=43349,769950,1075175
BC00290=41321,769954,1075175
BC00291=41321,769954,1075175
BC00292=41321,769954,1075175
BC00293=35772,778392,1075175
BC00294=49239,757053,1075175
BC00295=43736,767232,1075175
BC00296=44978,768291,1075175
BC00297=48083,770938,1075175
BC00298=48062,770936,1075175
BC00299=32781,783617,1075175
BC00300=28001,752077,1075175
BC00301=28012,752078,1075175
BC00302=32603,757759,1075175
BC00303=34440,760032,1075175
BC00304=34440,760032,1075175
BC00305=34440,760032,1075175
BC00306=31354,801365,1075175
BC00307=31607,741816,1075175
BC00308=33541,764942,1075175
BC00309=31586,765733,1075175
BC00310=26698,767709,1075175
BC00311=181441,722385,1075175
BC00312=206367,695978,993979
BC00313=43511,699656,343050
BC00314=15,700638,169199
BC00315=15,700638,169199
BC00316=15,702258,154627
BC00317=15,702907,148798
BC00318=15,702907,148798
BC00319=15,702907,148798
BC00320=15,695953,159545
BC00321=15,692250,164622
BC00322=15,689364,165916
BC00323=15,687048,165746
BC00324=15,688612,165744
BC00325=15,682519,161681
BC00326=15,683515,161688
BC00327=15,685058,161698
BC00328=15,689706,161726
BC00329=15,691438,161737
BC00330=15,696374,161765
BC00331=15,698216,161776
BC00332=15,700511,161790
BC00333=15,706376,161888
BC00334=15,705589,161798
BC00335=15,703851,169282
BC00336=15,699507,187994
BC00337=15,709054,229408
BC00338=15,696835,229408
BC00339=302372,698952,211490
BC00340=302372,717858,201268
BC00341=302372,750216,183774
BC00342=302372,750216,53
BC00343=302410,756221,53
BC00344=302425,758623,53
BC00345=302425,758623,53
BC00346=302425,758623,53
BC00347=299311,758688,53
BC00348=290325,759252,53
BC00349=285447,760748,53
BC00350=288289,760789,53
BC00351=287404,761796,53
BC00352=282605,764489,53
BC00353=263685,776785,53
BC00354=261483,775366,53
BC00355=255977,771818,53
BC00356=293911,751455,53
BC00357=295135,757520,53
BC00358=295624,759946,53
BC00359=295624,759946,53
BC00360=295624,759946,53
BC00361=272885,771858,53
BC00362=277126,769514,53
BC00363=254622,787284,53
BC00364=252160,786227,53
BC00365=246006,783585,53
BC00366=355967,746549,7296
BC00367=398174,732333,10075
BC00368=398174,732336,53
BC00369=398174,726917,53
BC00370=398174,724749,53
BC00371=398174,724749,53
BC00372=398174,724749,53
BC00373=398174,724759,53
BC00374=398174,724912,53
BC00375=398174,724618,53
BC00376=398174,726661,53
BC00377=398174,731768,53
BC00378=368426,774050,236358
BC00379=368302,768625,217333
BC00380=368253,766455,209723
BC00381=368253,766455,209723
BC00382=368253,766455,209723
BC00383=361154,766186,208862
BC00384=362122,766486,208257
BC00385=355834,766353,203745
BC00386=355004,768447,211098
BC00387=352929,773681,229482
BC00388=352908,773678,283249
BC00389=390912,664927,107315
BC00390=390215,665602,80639
BC00391=389936,665872,69969
BC00392=389936,665872,69969
BC00393=389936,665872,69969
BC00394=389934,666486,69971
BC00395=390213,666216,80641
BC00396=390910,665541,107318
BC00397=398174,768127,53
BC00398=398174,762708,53
BC00399=398174,760540,53
BC00400=398174,760540,53
BC00401=398174,760540,53
BC00402=398174,760550,53
BC00403=398174,760703,53
BC00404=398174,760409,53
BC00405=398174,762452,53
BC00406=398174,767558,53
BC00407=368308,809841,236482
BC00408=368184,804416,217457
BC00409=368134,802246,209847
BC00410=368134,802246,209847
BC00411=368134,802246,209847
BC00412=361036,801977,208986
BC00413=362004,802277,208380
BC00414=355716,802144,203868
BC00415=354886,804238,211222
BC00416=352810,809472,229606
BC00417=352790,809469,283373
BC00418=390793,700718,107439
BC00419=390096,701392,80763
BC00420=389818,701662,70092
BC00421=389818,701662,70092
BC00422=389818,701662,70092
BC00423=389816,702277,70095
BC00424=390094,702007,80765
BC00425=390791,701332,107441
BC00426=398174,803918,53
BC00427=398174,798498,53
BC00428=398174,796331,53
BC00429=398174,796331,53
BC00430=398174,796331,53
BC00431=398174,796340,53
BC00432=398174,796494,53
BC00433=398174,796200,53
BC00434=398174,798243,53
BC00435=398174,803349,53
BC00436=379839,832243,68523
BC00437=379715,826818,49498
BC00438=379665,824648,41888
BC00439=379665,824648,41888
BC00440=379665,824648,41888
BC00441=372567,824379,41027
BC00442=373535,824679,40421
BC00443=367247,824546,35909
BC00444=366417,826640,43263
BC00445=364341,831874,61647
BC00446=364320,831871,115414
BC00447=390675,736509,107563
BC00448=389978,737183,80887
BC00449=389699,737453,70216
BC00450=389699,737453,70216
BC00451=389699,737453,70216
BC00452=389697,738068,70218
BC00453=389976,737798,80889
BC00454=390673,737123,107565
BC00455=390673,737123,107565
BC00456=390673,737123,107565
BC00457=390673,737123,107565
BC00458=290974,720775,160770
BC00459=290667,722939,153208
BC00460=290667,722939,153208
BC00461=290667,722939,153208
BC00462=263990,723128,151402
BC00463=263013,723888,154276
BC00464=239902,731218,144781
BC00465=238128,729410,151082
BC00466=283521,718621,232190
BC00467=282179,720936,226764
BC00468=282179,720936,226764
BC00469=282179,720936,226764
BC00470=283052,720936,222522
BC00471=284913,720944,213537
BC00472=285794,720952,209313
BC00473=287136,718637,214739
BC00474=259950,703583,235329
BC00475=279991,738060,276884
BC00476=280001,738061,250000
BC00477=280813,743470,231112
BC00478=281137,745634,223556
BC00479=281137,745634,223556
BC00480=281137,745634,223556
BC00481=273506,746410,219687
BC00482=271690,747489,222922
BC00483=250689,754377,213689
BC00484=248915,752569,219990
BC00485=244479,748048,235742
BC00486=244458,748045,289510
BC00487=271703,701029,53
BC00488=272027,703193,53
BC00489=272027,703193,53
BC00490=272027,703193,53
BC00491=266411,707508,53
BC00492=262746,705272,53
BC00493=244606,713601,53
BC00494=242832,711793,53
BC00495=238396,707272,53
BC00496=238375,707270,53
BC00497=68499,695430,53
BC00498=68499,694666,53
BC00499=15,702747,12011
BC00500=15,702747,12011
BC00501=15,702747,12011
BC00502=15,707131,53
BC00503=15,708885,53
BC00504=15,708885,53
BC00505=15,708885,53
BC00506=26435,696636,53
BC00507=24834,696972,53
BC00508=20144,697212,53
BC00509=12426,698694,53
BC00510=9188,699084,53
BC00511=6011,699829,53
BC00512=2457,701378,53
BC00513=15,701853,53
BC00514=237,702707,53
BC00515=266,702707,53
BC00516=554,700278,53
BC00517=1273,694207,10484
BC00518=15,702747,12011
BC00519=15,702747,12011
BC00520=297950,700262,21134
BC00521=297950,699644,21134
BC00522=367073,697623,223727
BC00523=363305,702964,209184
BC00524=361798,705100,203367
BC00525=361798,705100,203367
BC00526=361798,705100,203367
BC00527=362672,705098,199128
BC00528=364534,705107,190143
BC00529=365413,705116,185916
BC00530=366920,702980,191733
BC00531=370688,697639,206275
BC00532=282559,738406,156506
BC00533=278791,743746,141963
BC00534=277284,745883,136146
BC00535=277284,745883,136146
BC00536=277284,745883,136146
BC00537=278130,745881,132041
BC00538=280020,745889,122922
BC00539=280871,745899,118829
BC00540=282379,743762,124646
BC00541=286147,738422,139188
BC00542=286126,738419,192956
BC00543=299995,822903,82685
BC00544=302547,827772,63763
BC00545=303567,829720,56193
BC00546=303567,829720,56193
BC00547=303567,829720,56193
BC00548=313993,826328,55950
BC00549=299999,831192,55994
BC00550=295498,832741,55983
BC00551=295000,830612,63551
BC00552=293755,825289,82470
BC00553=284848,832154,53
BC00554=288620,836218,53
BC00555=290129,837843,53
BC00556=290129,837843,53
BC00557=290129,837843,53
BC00558=294114,835300,53
BC00559=305389,828088,53
BC00560=309368,825536,53
BC00561=307859,823910,53
BC00562=304087,819847,53
BC00563=304889,824233,171046
BC00564=304889,700105,171046
BC00565=83775,699365,9536
BC00566=83775,690394,164839
BC00567=83766,691735,138369
BC00568=83762,692272,127780
BC00569=83762,692272,127780
BC00570=83762,692272,127780
BC00571=83750,695878,127793
BC00572=83754,695342,138381
BC00573=83763,694001,164852
BC00574=83763,737347,138110
BC00575=83763,737347,138110
BC00576=197026,737412,62024
BC00577=197037,737414,35140
BC00578=197030,738091,8361
BC00579=197027,738361,53
BC00580=197027,738361,53
BC00581=197027,738361,53
BC00582=197015,741973,53
BC00583=197018,741702,8374
BC00584=197025,741025,35153
BC00585=196904,776946,35277
BC00586=196898,777623,8498
BC00587=196895,777893,53
BC00588=196895,777893,53
BC00589=196895,777893,53
BC00590=196883,781477,53
BC00591=196886,781207,8510
BC00592=196893,780530,35289
BC00593=196882,780528,62173
BC00594=171385,775077,62173
BC00595=211973,723981,24737
BC00596=211368,723652,53
BC00597=211126,723520,53
BC00598=211126,723520,53
BC00599=211126,723520,53
BC00600=207872,721695,53
BC00601=208114,721826,53
BC00602=208718,722155,24737
BC00603=205285,720250,53
BC00604=202926,718936,53
BC00605=201983,718411,53
BC00606=201983,718411,53
BC00607=201983,718411,53
BC00608=198706,716573,53
BC00609=199649,717098,53
BC00610=202008,718412,53
BC00611=190841,744312,53
BC00612=188482,742998,53
BC00613=187539,742473,53
BC00614=187539,742473,53
BC00615=187539,742473,53
BC00616=184322,740668,53
BC00617=185265,741194,53
BC00618=187624,742507,53
BC00619=211648,716653,11834
BC00620=209289,715339,53
BC00621=208346,714814,53
BC00622=208346,714814,53
BC00623=208346,714814,53
BC00624=205069,712976,53
BC00625=206012,713501,53
BC00626=208371,714815,11834
BC00627=184359,725138,114504
BC00628=155631,789719,177806
BC00629=155631,789719,177806
BC00630=155631,789719,177806
BC00631=155631,789719,177806
BC00632=155631,789719,177806
BC00633=155631,789719,177806
BC00634=155631,789719,177806
BC00635=155631,789719,177806
BC00636=155631,789719,177806
BC00637=155631,789719,177806
BC00638=155631,789719,177806
BC00639=151946,797646,240508
BC00640=151946,797646,240508
BC00641=151946,797646,240508
BC00642=151946,797646,240508
BC00643=151946,797646,240508
BC00644=151946,797646,240508
BC00645=151946,797646,240508
BC00646=151946,797646,240508
BC00647=151946,797646,240508
BC00648=151946,797646,240508
BC00649=151946,797646,240508
BC00650=164113,763380,121188
BC00651=164113,711732,121188
BC00652=279725,698376,121188
BC00653=279725,755875,121188
BC00654=373318,818673,338864
BC00655=378182,828617,343030
BC00656=370596,830533,347720
BC00657=367562,831300,349596
BC00658=367562,831300,349596
BC00659=367562,831300,349596
BC00660=367559,831304,333465
BC00661=367475,831445,53
BC00662=347960,827291,53
BC00663=350891,826549,53
BC00664=358219,824694,53
BC00665=350992,826871,341327
BC00666=342745,817956,297922
BC00667=331538,781751,238935
BC00668=337189,786996,243611
BC00669=339450,789094,245481
BC00670=339450,789094,245481
BC00671=339450,789094,245481
BC00672=339447,789098,229351
BC00673=339418,789147,54092
BC00674=339415,789152,37962
BC00675=337154,787054,36092
BC00676=331503,781810,31416
BC00677=331503,781810,310369
BC00678=331503,678865,310369
EC00000=798156,0
EC00001=798156,0
EC00002=798156,0
EC00003=798156,0
EC00004=798156,0
EC00005=798156,0
EC00006=798156,0
EC00007=798156,0
EC00008=798156,0
EC00009=798156,0
EC00010=798156,0
EC00011=798156,0
EC00012=798156,0
EC00013=798156,0
EC00014=798156,0
EC00015=798156,0
EC00016=798156,0
EC00017=798156,0
EC00018=798156,0
EC00019=798156,0
EC00020=798156,0
EC00021=798156,0
EC00022=798156,0
EC00023=798156,0
EC00024=798156,0
EC00025=798156,0
EC00026=798156,0
EC00027=798156,0
EC00028=798156,0
EC00029=798156,0
EC00030=798156,0
EC00031=798156,0
EC00032=798156,0
EC00033=798156,0
EC00034=798156,0
EC00035=798156,0
EC00036=798156,0
EC00037=798156,0
EC00038=798156,0
EC00039=798156,0
EC00040=798156,0
EC00041=798156,0
EC00042=798156,0
EC00043=798156,0
EC00044=798156,0
EC00045=798156,0
EC00046=798156,0
EC00047=798155,0
EC00048=798156,0
EC00049=798156,0
EC00050=798156,0
EC00051=798156,0
EC00052=798156,0
EC00053=798156,0
EC00054=798156,0
EC00055=798156,0
EC00056=798156,0
EC00057=798156,0
EC00058=798156,0
EC00059=798156,0
EC00060=798156,0
EC00061=798156,0
EC00062=798156,0
EC00063=798156,0
EC00064=798156,0
EC00065=798156,0
EC00066=798156,0
EC00067=798156,0
EC00068=798156,0
EC00069=798156,0
EC00070=798156,0
EC00071=798156,0
EC00072=798156,0
EC00073=798156,0
EC00074=798156,0
EC00075=798151,1
EC00076=798155,0
EC00077=798156,0
EC00078=798156,0
EC00079=798156,0
EC00080=798156,0
EC00081=798156,0
EC00082=798156,0
EC00083=798156,0
EC00084=798156,0
EC00085=798156,0
EC00086=798156,0
EC00087=798156,0
EC00088=798156,0
EC00089=798156,0
EC00090=798156,0
EC00091=798156,0
EC00092=798156,0
EC00093=798156,0
EC00094=798156,0
EC00095=798156,0
EC00096=798156,0
EC00097=798156,0
EC00098=798156,0
EC00099=798156,0
EC00100=798156,0
EC00101=798156,0
EC00102=798156,0
EC00103=798156,0
EC00104=798156,0
EC00105=798156,0
EC00106=798156,0
EC00107=798156,0
EC00108=798156,0
EC00109=798156,0
EC00110=798156,0
EC00111=798156,0
EC00112=798156,0
EC00113=798156,0
EC00114=798156,0
EC00115=798156,0
EC00116=798156,0
EC00117=798156,0
EC00118=798156,0
EC00119=798156,0
EC00120=798156,0
EC00121=798156,0
EC00122=798156,0
EC00123=798156,0
EC00124=798156,0
EC00125=798156,0
EC00126=798156,0
EC00127=798156,0
EC00128=798156,0
EC00129=798156,0
EC00130=798156,0
EC00131=798156,0
EC00132=798156,0
EC00133=798156,0
EC00134=798156,0
EC00135=798156,0
EC00136=798156,0
EC00137=798156,0
EC00138=798156,0
EC00139=798156,0
EC00140=798156,0
EC00141=798156,0
EC00142=798156,0
EC00143=798156,0
EC00144=798156,0
EC00145=821191,0
EC00146=883374,0
EC00147=975524,0
EC00148=975524,0
EC00149=975524,0
EC00150=975524,0
EC00151=975524,0
EC00152=975524,0
EC00153=975524,0
EC00154=975524,0
EC00155=975524,0
EC00156=975524,0
EC00157=975524,0
EC00158=975524,0
EC00159=975524,0
EC00160=975524,0
EC00161=975524,0
EC00162=975524,0
EC00163=975524,0
EC00164=975524,0
EC00165=975524,0
EC00166=975524,0
EC00167=975524,0
EC00168=975524,0
EC00169=975524,0
EC00170=975524,0
EC00171=975524,0
EC00172=975524,0
EC00173=975524,0
EC00174=975524,0
EC00175=975524,0
EC00176=975524,0
EC00177=975524,0
EC00178=975524,0
EC00179=975524,0
EC00180=975524,0
EC00181=975524,0
EC00182=975524,0
EC00183=975524,0
EC00184=975524,0
EC00185=975524,0
EC00186=975524,0
EC00187=975524,0
EC00188=975524,0
EC00189=975524,0
EC00190=975524,0
EC00191=975524,0
EC00192=975524,0
EC00193=975524,0
EC00194=975524,0
EC00195=975524,0
EC00196=975524,0
EC00197=975524,0
EC00198=975524,0
EC00199=975524,0
EC00200=975524,0
EC00201=975524,0
EC00202=975524,0
EC00203=975524,0
EC00204=975524,0
EC00205=975524,0
EC00206=975524,0
EC00207=975524,0
EC00208=975524,0
EC00209=975524,0
EC00210=975524,0
EC00211=975524,0
EC00212=975524,0
EC00213=975524,0
EC00214=975524,0
EC00215=975524,0
EC00216=975524,0
EC00217=975524,0
EC00218=975524,0
EC00219=975524,0
EC00220=975524,0
EC00221=975524,0
EC00222=975524,0
EC00223=975524,0
EC00224=975524,0
EC00225=975524,0
EC00226=975524,0
EC00227=975524,0
EC00228=975524,0
EC00229=975524,0
EC00230=975524,0
EC00231=975524,0
EC00232=975524,0
EC00233=975524,0
EC00234=975524,0
EC00235=975524,0
EC00236=975524,0
EC00237=975524,0
EC00238=975524,0
EC00239=975524,0
EC00240=975524,0
EC00241=975524,0
EC00242=975524,0
EC00243=975524,0
EC00244=975524,0
EC00245=975524,0
EC00246=975524,0
EC00247=975524,0
EC00248=975524,0
EC00249=975524,0
EC00250=975524,0
EC00251=975524,0
EC00252=975524,0
EC00253=975524,0
EC00254=975524,0
EC00255=975524,0
EC00256=975524,0
EC00257=975524,0
EC00258=975524,0
EC00259=975524,0
EC00260=975524,0
EC00261=975524,0
EC00262=975524,0
EC00263=975524,0
EC00264=975524,0
EC00265=975524,0
EC00266=975524,0
EC00267=975524,0
EC00268=975524,0
EC00269=975524,0
EC00270=975524,0
EC00271=975524,0
EC00272=975524,0
EC00273=975524,0
EC00274=975524,0
EC00275=975524,0
EC00276=975524,0
EC00277=975524,0
EC00278=975524,0
EC00279=975524,0
EC00280=975524,0
EC00281=975524,0
EC00282=975524,0
EC00283=975524,0
EC00284=975524,0
EC00285=975524,0
EC00286=975524,0
EC00287=975524,0
EC00288=975524,0
EC00289=975524,0
EC00290=975524,0
EC00291=975524,0
EC00292=975524,0
EC00293=975524,0
EC00294=975524,0
EC00295=975524,0
EC00296=975524,0
EC00297=975524,0
EC00298=975524,0
EC00299=975524,0
EC00300=975524,0
EC00301=975524,0
EC00302=975524,0
EC00303=975524,0
EC00304=975524,0
EC00305=975524,0
EC00306=975524,0
EC00307=975524,0
EC00308=975524,0
EC00309=975524,0
EC00310=975524,0
EC00311=975524,0
EC00312=959628,0
EC00313=832192,0
EC00314=798156,0
EC00315=798156,0
EC00316=798156,0
EC00317=798156,0
EC00318=798156,0
EC00319=798156,0
EC00320=798156,0
EC00321=798156,0
EC00322=798156,0
EC00323=798156,0
EC00324=798156,0
EC00325=798156,0
EC00326=798156,0
EC00327=798156,0
EC00328=798156,0
EC00329=798156,0
EC00330=798156,0
EC00331=798156,0
EC00332=798156,0
EC00333=798156,0
EC00334=798156,0
EC00335=798156,0
EC00336=798156,0
EC00337=798156,0
EC00338=798156,0
EC00339=798156,0
EC00340=798156,0
EC00341=798156,0
EC00342=798156,0
EC00343=798156,0
EC00344=798156,0
EC00345=798156,0
EC00346=798156,0
EC00347=798156,0
EC00348=798156,0
EC00349=798156,0
EC00350=798156,0
EC00351=798156,0
EC00352=798156,0
EC00353=798156,0
EC00354=798156,0
EC00355=798156,0
EC00356=798156,0
EC00357=798156,0
EC00358=798156,0
EC00359=798156,0
EC00360=798156,0
EC00361=798156,0
EC00362=798156,0
EC00363=798156,0
EC00364=798156,0
EC00365=798156,0
EC00366=798156,0
EC00367=798156,0
EC00368=798156,0
EC00369=798156,0
EC00370=798156,0
EC00371=798156,0
EC00372=798156,0
EC00373=798156,0
EC00374=798156,0
EC00375=798156,0
EC00376=798156,0
EC00377=798156,0
EC00378=798156,0
EC00379=798156,0
EC00380=798156,0
EC00381=798156,0
EC00382=798156,0
EC00383=798156,0
EC00384=798156,0
EC00385=798156,0
EC00386=798156,0
EC00387=798156,0
EC00388=798156,0
EC00389=798156,0
EC00390=798156,0
EC00391=798156,0
EC00392=798156,0
EC00393=798156,0
EC00394=798156,0
EC00395=798156,0
EC00396=798156,0
EC00397=798156,0
EC00398=798156,0
EC00399=798156,0
EC00400=798156,0
EC00401=798156,0
EC00402=798156,0
EC00403=798156,0
EC00404=798156,0
EC00405=798156,0
EC00406=798156,0
EC00407=798156,0
EC00408=798156,0
EC00409=798156,0
EC00410=798156,0
EC00411=798156,0
EC00412=798156,0
EC00413=798156,0
EC00414=798156,0
EC00415=798156,0
EC00416=798156,0
EC00417=798156,0
EC00418=798156,0
EC00419=798156,0
EC00420=798156,0
EC00421=798156,0
EC00422=798156,0
EC00423=798156,0
EC00424=798156,0
EC00425=798156,0
EC00426=798156,0
EC00427=798156,0
EC00428=798156,0
EC00429=798156,0
EC00430=798156,0
EC00431=798156,0
EC00432=798156,0
EC00433=798156,0
EC00434=798156,0
EC00435=798156,0
EC00436=798156,0
EC00437=798156,0
EC00438=798156,0
EC00439=798156,0
EC00440=798156,0
EC00441=798156,0
EC00442=798156,0
EC00443=798156,0
EC00444=798156,0
EC00445=798156,0
EC00446=798156,0
EC00447=798156,0
EC00448=798156,0
EC00449=798156,0
EC00450=798156,0
EC00451=798156,0
EC00452=798156,0
EC00453=798156,0
EC00454=798156,0
EC00455=798156,0
EC00456=798156,0
EC00457=798156,0
EC00458=798156,0
EC00459=798156,0
EC00460=798156,0
EC00461=798156,0
EC00462=798156,0
EC00463=798156,0
EC00464=798156,0
EC00465=798156,0
EC00466=798156,0
EC00467=798156,0
EC00468=798156,0
EC00469=798156,0
EC00470=798156,0
EC00471=798156,0
EC00472=798156,0
EC00473=798156,0
EC00474=798156,0
EC00475=798156,0
EC00476=798156,0
EC00477=798156,0
EC00478=798156,0
EC00479=798156,0
EC00480=798156,0
EC00481=798156,0
EC00482=798156,0
EC00483=798156,0
EC00484=798156,0
EC00485=798156,0
EC00486=798156,0
EC00487=798156,0
EC00488=798156,0
EC00489=798156,0
EC00490=798156,0
EC00491=798156,0
EC00492=798156,0
EC00493=798156,0
EC00494=798156,0
EC00495=798156,0
EC00496=798156,0
EC00497=798156,0
EC00498=798156,0
EC00499=798156,0
EC00500=798156,0
EC00501=798156,0
EC00502=798156,0
EC00503=798156,0
EC00504=798156,0
EC00505=798156,0
EC00506=798156,0
EC00507=798156,0
EC00508=798156,0
EC00509=798156,0
EC00510=798156,0
EC00511=798156,0
EC00512=798156,0
EC00513=798156,0
EC00514=798156,0
EC00515=798156,0
EC00516=798156,0
EC00517=798156,0
EC00518=798156,0
EC00519=798156,0
EC00520=798156,0
EC00521=798156,0
EC00522=798156,0
EC00523=798156,0
EC00524=798156,0
EC00525=798156,0
EC00526=798156,0
EC00527=798156,0
EC00528=798156,0
EC00529=798156,0
EC00530=798156,0
EC00531=798156,0
EC00532=798156,0
EC00533=798156,0
EC00534=798156,0
EC00535=798156,0
EC00536=798156,0
EC00537=798156,0
EC00538=798156,0
EC00539=798156,0
EC00540=798156,0
EC00541=798156,0
EC00542=798156,0
EC00543=798156,0
EC00544=798156,0
EC00545=798156,0
EC00546=798156,0
EC00547=798156,0
EC00548=798156,0
EC00549=798156,0
EC00550=798156,0
EC00551=798156,0
EC00552=798156,0
EC00553=798156,0
EC00554=798156,0
EC00555=798156,0
EC00556=798156,0
EC00557=798156,0
EC00558=798156,0
EC00559=798156,0
EC00560=798156,0
EC00561=798156,0
EC00562=798156,0
EC00563=798156,0
EC00564=798156,0
EC00565=798156,0
EC00566=798156,0
EC00567=798156,0
EC00568=798156,0
EC00569=798156,0
EC00570=798156,0
EC00571=798156,0
EC00572=798156,0
EC00573=798156,0
EC00574=798156,0
EC00575=798156,0
EC00576=798156,0
EC00577=798156,0
EC00578=798156,0
EC00579=798156,0
EC00580=798156,0
EC00581=798156,0
EC00582=798156,0
EC00583=798156,0
EC00584=798156,0
EC00585=798156,0
EC00586=798156,0
EC00587=798156,0
EC00588=798156,0
EC00589=798156,0
EC00590=798156,0
EC00591=798156,0
EC00592=798156,0
EC00593=798156,0
EC00594=798156,0
EC00595=798156,0
EC00596=798156,0
EC00597=798156,0
EC00598=798156,0
EC00599=798156,0
EC00600=798156,0
EC00601=798156,0
EC00602=798156,0
EC00603=798156,0
EC00604=798156,0
EC00605=798156,0
EC00606=798156,0
EC00607=798156,0
EC00608=798156,0
EC00609=798156,0
EC00610=798156,0
EC00611=798156,0
EC00612=798156,0
EC00613=798156,0
EC00614=798156,0
EC00615=798156,0
EC00616=798156,0
EC00617=798156,0
EC00618=798156,0
EC00619=798156,0
EC00620=798156,0
EC00621=798156,0
EC00622=798156,0
EC00623=798156,0
EC00624=798156,0
EC00625=798156,0
EC00626=798156,0
EC00627=798156,0
EC00628=798156,0
EC00629=798156,0
EC00630=798156,0
EC00631=798156,0
EC00632=798156,0
EC00633=798156,0
EC00634=798156,0
EC00635=798156,0
EC00636=798156,0
EC00637=798156,0
EC00638=798156,0
EC00639=798156,0
EC00640=798156,0
EC00641=798156,0
EC00642=798156,0
EC00643=798156,0
EC00644=798156,0
EC00645=798156,0
EC00646=798156,0
EC00647=798156,0
EC00648=798156,0
EC00649=798156,0
EC00650=798156,0
EC00651=798156,0
EC00652=798156,0
EC00653=798156,0
EC00654=798156,0
EC00655=798156,0
EC00656=798156,0
EC00657=798156,0
EC00658=798156,0
EC00659=798156,0
EC00660=798156,0
EC00661=798156,0
EC00662=798156,0
EC00663=798156,0
EC00664=798156,0
EC00665=798156,0
EC00666=798156,0
EC00667=798156,0
EC00668=798156,0
EC00669=798156,0
EC00670=798156,0
EC00671=798156,0
EC00672=798156,0
EC00673=798156,0
EC00674=798156,0
EC00675=798156,0
EC00676=798156,0
EC00677=798156,0
EC00678=798156,0
///POSTYPE BASE
///RECTAN
///RCONF 0,0,0,0,0,0,0,0,0,0,0,0,0,0,0,0,0,0,0,0,0,0,0,0
P00006=0.222,-3.123,-1.508,0.0000,0.0000,0.0000
P00021=-0.225,-6.128,-0.405,0.0000,0.0000,0.0000
P00022=0.222,-3.123,-1.508,0.0000,0.0000,0.0000
P00023=0.143,-0.036,0.682,0.0000,0.0000,0.0000
P00024=0.145,-0.552,1.326,0.0000,0.0000,0.0000
P00025=-2.003,0.006,0.728,0.0000,0.0000,0.0000
P00026=0.562,-0.002,-0.337,0.0000,0.0000,0.0000
P00027=-0.746,0.015,-9.096,0.0000,0.0000,0.0000
P00028=-2.237,-0.018,-7.702,0.0000,0.0000,0.0000
P00029=-2.156,-0.086,-4.681,0.0000,0.0000,0.0000
P00030=5.926,-4.294,-1.390,0.0000,0.0000,0.0000
P00031=1.853,-0.001,-1.549,0.0000,0.0000,0.0000
P00032=1.957,0.503,-7.217,0.0000,0.0000,0.0000
P00041=0.192,3.924,0.305,0.0000,0.0000,0.0000
P00042=-0.217,1.941,0.413,0.0000,0.0000,0.0000
P00043=-0.044,-1.937,1.197,0.0000,0.0000,0.0000
P00044=0.687,-2.322,1.156,0.0000,0.0000,0.0000
P00045=-0.068,-0.810,1.603,0.0000,0.0000,0.0000
P00046=0.799,0.043,1.292,0.0000,0.0000,0.0000
//INST
///DATE 2024/01/08 19:41
///ATTR SC,RW
///GROUP1 RB1,BS1
///GROUP2 ST1
NOP
'OK_r2_O57-69(1)(90,0)
'Down
'Path S1900
SFTOF3D
MOVJ C00000 BC00000 VJ=100.00  +MOVJ EC00000 VJ=100.00
MOVL C00001 BC00001 V=100.0  +MOVJ EC00001 VJ=100.00
SMOVL C00002 BC00002 V=60.0  +MOVJ EC00002
SREFP 3 C00003 BC00003  +REFP EC00003
CALL JOB:SEARCH-R1-S13D
SET P031 P006
SFTON3D P031
SMOVL C00004 BC00004 V=60.0  +MOVJ EC00004
SMOVL C00005 BC00005 V=60.0  +MOVJ EC00005
SREFP 3 C00006 BC00006  +REFP EC00006
CALL JOB:SEARCH-R1-S13D
SET P031 P006
SFTON3D P031
SMOVL C00007 BC00007 V=60.0  +MOVJ EC00007
MOVL C00008 BC00008 V=400.0  +MOVJ EC00008 VJ=100.00
MOVL C00009 BC00009 V=1000.0  +MOVJ EC00009 VJ=100.00
'Path S1901
SFTOF3D
PAUSE
MOVJ C00010 BC00010 VJ=100.00  +MOVJ EC00010 VJ=100.00
MOVJ C00011 BC00011 VJ=100.00  +MOVJ EC00011 VJ=100.00
MOVL C00012 BC00012 V=100.0  +MOVJ EC00012 VJ=100.00
SMOVL C00013 BC00013 V=60.0  +MOVJ EC00013
SREFP 3 C00014 BC00014  +REFP EC00014
CALL JOB:SEARCH-R1-S13D
SET P026 P006
SFTON3D P026
SMOVL C00015 BC00015 V=60.0  +MOVJ EC00015
SMOVL C00016 BC00016 V=60.0  +MOVJ EC00016
SREFP 3 C00017 BC00017  +REFP EC00017
CALL JOB:SEARCH-R1-S13D
SET P026 P006
SFTON3D P026
SMOVL C00018 BC00018 V=60.0  +MOVJ EC00018
MOVL C00019 BC00019 V=400.0  +MOVJ EC00019 VJ=100.00
MOVL C00020 BC00020 V=1000.0  +MOVJ EC00020 VJ=100.00
'Path S1902
SFTOF3D
MOVJ C00021 BC00021 VJ=100.00  +MOVJ EC00021 VJ=100.00
MOVL C00022 BC00022 V=100.0  +MOVJ EC00022 VJ=100.00
SMOVL C00023 BC00023 V=60.0  +MOVJ EC00023
SREFP 3 C00024 BC00024  +REFP EC00024
CALL JOB:SEARCH-R1-S13D
SET P027 P006
SFTON3D P027
SMOVL C00025 BC00025 V=60.0  +MOVJ EC00025
SMOVL C00026 BC00026 V=60.0  +MOVJ EC00026
SREFP 3 C00027 BC00027  +REFP EC00027
CALL JOB:SEARCH-R1-S13D
SET P027 P006
SFTON3D P027
SMOVL C00028 BC00028 V=60.0  +MOVJ EC00028
MOVL C00029 BC00029 V=400.0  +MOVJ EC00029 VJ=100.00
MOVL C00030 BC00030 V=1000.0  +MOVJ EC00030 VJ=100.00
'Path S1903
SFTOF3D
PAUSE
MOVJ C00031 BC00031 VJ=100.00  +MOVJ EC00031 VJ=100.00
MOVJ C00032 BC00032 VJ=100.00  +MOVJ EC00032 VJ=100.00
MOVL C00033 BC00033 V=100.0  +MOVJ EC00033 VJ=100.00
SMOVL C00034 BC00034 V=60.0  +MOVJ EC00034
SREFP 3 C00035 BC00035  +REFP EC00035
CALL JOB:SEARCH-R1-S13D
SET P022 P006
SFTON3D P022
SMOVL C00036 BC00036 V=60.0  +MOVJ EC00036
SMOVL C00037 BC00037 V=60.0  +MOVJ EC00037
SREFP 3 C00038 BC00038  +REFP EC00038
CALL JOB:SEARCH-R1-S13D
SET P022 P006
SFTON3D P022
SMOVL C00039 BC00039 V=60.0  +MOVJ EC00039
MOVL C00040 BC00040 V=400.0  +MOVJ EC00040 VJ=100.00
MOVL C00041 BC00041 V=1000.0  +MOVJ EC00041 VJ=100.00
MOVJ C00042 BC00042 VJ=100.00  +MOVJ EC00042 VJ=100.00
'Path S1904
SFTOF3D
PAUSE
MOVJ C00043 BC00043 VJ=100.00  +MOVJ EC00043 VJ=100.00
MOVJ C00044 BC00044 VJ=100.00  +MOVJ EC00044 VJ=100.00
MOVL C00045 BC00045 V=400.0  +MOVJ EC00045 VJ=100.00
SMOVL C00046 BC00046 V=60.0  +MOVJ EC00046
SREFP 3 C00047 BC00047  +REFP EC00047
CALL JOB:SEARCH-R1-S13D
SET P028 P006
SFTON3D P028
SMOVL C00048 BC00048 V=60.0  +MOVJ EC00048
SMOVL C00049 BC00049 V=60.0  +MOVJ EC00049
SREFP 3 C00050 BC00050  +REFP EC00050
CALL JOB:SEARCH-R1-S13D
SET P028 P006
SFTON3D P028
SMOVL C00051 BC00051 V=60.0  +MOVJ EC00051
MOVL C00052 BC00052 V=400.0  +MOVJ EC00052 VJ=100.00
MOVL C00053 BC00053 V=1000.0  +MOVJ EC00053 VJ=100.00
'Path S1905
SFTOF3D
PAUSE
MOVJ C00054 BC00054 VJ=100.00  +MOVJ EC00054 VJ=100.00
SMOVL C00055 BC00055 V=60.0  +MOVJ EC00055
SREFP 3 C00056 BC00056  +REFP EC00056
CALL JOB:SEARCH-R1-S13D
SET P029 P006
SFTON3D P029
SMOVL C00057 BC00057 V=60.0  +MOVJ EC00057
SMOVL C00058 BC00058 V=60.0  +MOVJ EC00058
SREFP 3 C00059 BC00059  +REFP EC00059
CALL JOB:SEARCH-R1-S13D
SET P029 P006
SFTON3D P029
SMOVL C00060 BC00060 V=60.0  +MOVJ EC00060
MOVL C00061 BC00061 V=400.0  +MOVJ EC00061 VJ=100.00
MOVL C00062 BC00062 V=1000.0  +MOVJ EC00062 VJ=100.00
'Path S1906
SFTOF3D
PAUSE
MOVJ C00063 BC00063 VJ=100.00  +MOVJ EC00063 VJ=100.00
MOVL C00064 BC00064 V=100.0  +MOVJ EC00064 VJ=100.00
SMOVL C00065 BC00065 V=60.0  +MOVJ EC00065
SREFP 3 C00066 BC00066  +REFP EC00066
CALL JOB:SEARCH-R1-S13D
SET P030 P006
SFTON3D P030
SMOVL C00067 BC00067 V=60.0  +MOVJ EC00067
SMOVL C00068 BC00068 V=60.0  +MOVJ EC00068
SREFP 3 C00069 BC00069  +REFP EC00069
CALL JOB:SEARCH-R1-S13D
SET P030 P006
SFTON3D P030
SMOVL C00070 BC00070 V=60.0  +MOVJ EC00070
MOVL C00071 BC00071 V=400.0  +MOVJ EC00071 VJ=100.00
MOVL C00072 BC00072 V=1000.0  +MOVJ EC00072 VJ=100.00
MOVJ C00073 BC00073 VJ=100.00  +MOVJ EC00073 VJ=100.00
MOVJ C00074 BC00074 VJ=100.00  +MOVJ EC00074 VJ=100.00
MOVJ C00075 BC00075 VJ=100.00  +MOVJ EC00075 VJ=100.00
'Path S1907
SFTOF3D
PAUSE
MOVJ C00076 BC00076 VJ=100.00  +MOVJ EC00076 VJ=100.00  //MP
MOVL C00077 BC00077 V=400.0  +MOVJ EC00077 VJ=100.00
SMOVL C00078 BC00078 V=60.0  +MOVJ EC00078
SREFP 3 C00079 BC00079  +REFP EC00079
CALL JOB:SEARCH-R1-S13D
SET P023 P006
SFTON3D P023
SMOVL C00080 BC00080 V=60.0  +MOVJ EC00080
SMOVL C00081 BC00081 V=60.0  +MOVJ EC00081
SREFP 3 C00082 BC00082  +REFP EC00082
CALL JOB:SEARCH-R1-S13D
SET P023 P006
SFTON3D P023
SMOVL C00083 BC00083 V=60.0  +MOVJ EC00083
SMOVL C00084 BC00084 V=60.0  +MOVJ EC00084
SREFP 3 C00085 BC00085  +REFP EC00085
CALL JOB:SEARCH-R1-S13D
SET P023 P006
SFTON3D P023
SMOVL C00086 BC00086 V=60.0  +MOVJ EC00086
MOVL C00087 BC00087 V=400.0  +MOVJ EC00087 VJ=100.00
MOVL C00088 BC00088 V=1000.0  +MOVJ EC00088 VJ=100.00
MOVL C00089 BC00089 V=1000.0  +MOVJ EC00089 VJ=100.00
MOVJ C00090 BC00090 VJ=100.00  +MOVJ EC00090 VJ=100.00
'Path S1908
SFTOF3D
MOVL C00091 BC00091 V=400.0  +MOVJ EC00091 VJ=100.00
SMOVL C00092 BC00092 V=60.0  +MOVJ EC00092
SREFP 3 C00093 BC00093  +REFP EC00093
CALL JOB:SEARCH-R1-S13D
SET P024 P006
SFTON3D P024
SMOVL C00094 BC00094 V=60.0  +MOVJ EC00094
SMOVL C00095 BC00095 V=60.0  +MOVJ EC00095
SREFP 3 C00096 BC00096  +REFP EC00096
CALL JOB:SEARCH-R1-S13D
SET P024 P006
SFTON3D P024
SMOVL C00097 BC00097 V=60.0  +MOVJ EC00097
SMOVL C00098 BC00098 V=60.0  +MOVJ EC00098
SREFP 3 C00099 BC00099  +REFP EC00099
CALL JOB:SEARCH-R1-S13D
SET P024 P006
SFTON3D P024
SMOVL C00100 BC00100 V=60.0  +MOVJ EC00100
MOVL C00101 BC00101 V=400.0  +MOVJ EC00101 VJ=100.00
MOVL C00102 BC00102 V=1000.0  +MOVJ EC00102 VJ=100.00
MOVL C00103 BC00103 V=1000.0  +MOVJ EC00103 VJ=100.00
'Path S1909
SFTOF3D
MOVJ C00104 BC00104 VJ=100.00  +MOVJ EC00104 VJ=100.00
MOVL C00105 BC00105 V=400.0  +MOVJ EC00105 VJ=100.00
SMOVL C00106 BC00106 V=60.0  +MOVJ EC00106
SREFP 3 C00107 BC00107  +REFP EC00107
CALL JOB:SEARCH-R1-S13D
SET P025 P006
SFTON3D P025
SMOVL C00108 BC00108 V=60.0  +MOVJ EC00108
SMOVL C00109 BC00109 V=60.0  +MOVJ EC00109
SREFP 3 C00110 BC00110  +REFP EC00110
CALL JOB:SEARCH-R1-S13D
SET P025 P006
SFTON3D P025
SMOVL C00111 BC00111 V=60.0  +MOVJ EC00111
SMOVL C00112 BC00112 V=60.0  +MOVJ EC00112
SREFP 3 C00113 BC00113  +REFP EC00113
CALL JOB:SEARCH-R1-S13D
SET P025 P006
SFTON3D P025
SMOVL C00114 BC00114 V=60.0  +MOVJ EC00114
MOVL C00115 BC00115 V=400.0  +MOVJ EC00115 VJ=100.00
MOVL C00116 BC00116 V=1000.0  +MOVJ EC00116 VJ=100.00
MOVL C00117 BC00117 V=1000.0  +MOVJ EC00117 VJ=100.00
MOVJ C00118 BC00118 VJ=100.00  +MOVJ EC00118 VJ=100.00
MOVJ C00119 BC00119 VJ=100.00  +MOVJ EC00119 VJ=100.00
MOVJ C00120 BC00120 VJ=100.00  +MOVJ EC00120 VJ=100.00
'Path S1910
SFTOF3D
MOVL C00121 BC00121 V=100.0  +MOVJ EC00121 VJ=100.00
SMOVL C00122 BC00122 V=60.0  +MOVJ EC00122
SREFP 3 C00123 BC00123  +REFP EC00123
CALL JOB:SEARCH-R1-S13D
SET P021 P006
SFTON3D P021
SMOVL C00124 BC00124 V=60.0  +MOVJ EC00124
SMOVL C00125 BC00125 V=60.0  +MOVJ EC00125
SREFP 3 C00126 BC00126  +REFP EC00126
CALL JOB:SEARCH-R1-S13D
SET P021 P006
SFTON3D P021
SMOVL C00127 BC00127 V=60.0  +MOVJ EC00127
SMOVL C00128 BC00128 V=60.0  +MOVJ EC00128
SREFP 3 C00129 BC00129  +REFP EC00129
CALL JOB:SEARCH-R1-S13D
SET P021 P006
SFTON3D P021
SMOVL C00130 BC00130 V=60.0  +MOVJ EC00130
MOVL C00131 BC00131 V=400.0  +MOVJ EC00131 VJ=100.00
MOVJ C00132 BC00132 VJ=100.00  +MOVJ EC00132 VJ=100.00
MOVJ C00133 BC00133 VJ=100.00  +MOVJ EC00133 VJ=100.00
MOVJ C00134 BC00134 VJ=100.00  +MOVJ EC00134 VJ=100.00
'Path S1912
SFTOF3D
MOVJ C00135 BC00135 VJ=100.00  +MOVJ EC00135 VJ=100.00
MOVL C00136 BC00136 V=400.0  +MOVJ EC00136 VJ=100.00
SMOVL C00137 BC00137 V=60.0  +MOVJ EC00137
SREFP 3 C00138 BC00138  +REFP EC00138
CALL JOB:SEARCH-R1-S13D
SET P032 P006
SFTON3D P032
SMOVL C00139 BC00139 V=60.0  +MOVJ EC00139
SMOVL C00140 BC00140 V=60.0  +MOVJ EC00140
SREFP 3 C00141 BC00141  +REFP EC00141
CALL JOB:SEARCH-R1-S13D
SET P032 P006
SFTON3D P032
SMOVL C00142 BC00142 V=60.0  +MOVJ EC00142
MOVL C00143 BC00143 V=400.0  +MOVJ EC00143 VJ=100.00
MOVL C00144 BC00144 V=1000.0  +MOVJ EC00144 VJ=100.00
'Up
MOVJ C00145 BC00145 VJ=100.00  +MOVJ EC00145 VJ=100.00
MOVJ C00146 BC00146 VJ=100.00  +MOVJ EC00146 VJ=100.00
MOVJ C00147 BC00147 VJ=100.00  +MOVJ EC00147 VJ=100.00
MOVJ C00148 BC00148 VJ=100.00  +MOVJ EC00148 VJ=100.00
'Path S1137
SFTOF3D
MOVJ C00149 BC00149 VJ=100.00  +MOVJ EC00149 VJ=100.00
MOVL C00150 BC00150 V=400.0  +MOVJ EC00150 VJ=100.00
SMOVL C00151 BC00151 V=60.0  +MOVJ EC00151
SREFP 3 C00152 BC00152  +REFP EC00152
CALL JOB:SEARCH-R1-S13D
SET P046 P006
SFTON3D P046
SMOVL C00153 BC00153 V=60.0  +MOVJ EC00153
SMOVL C00154 BC00154 V=60.0  +MOVJ EC00154
SREFP 3 C00155 BC00155  +REFP EC00155
CALL JOB:SEARCH-R1-S13D
SET P046 P006
SFTON3D P046
SMOVL C00156 BC00156 V=60.0  +MOVJ EC00156
MOVL C00157 BC00157 V=400.0  +MOVJ EC00157 VJ=100.00
MOVL C00158 BC00158 V=1000.0  +MOVJ EC00158 VJ=100.00
'Path S1169
SFTOF3D
MOVJ C00159 BC00159 VJ=100.00  +MOVJ EC00159 VJ=100.00
MOVL C00160 BC00160 V=400.0  +MOVJ EC00160 VJ=100.00
SMOVL C00161 BC00161 V=60.0  +MOVJ EC00161
SREFP 3 C00162 BC00162  +REFP EC00162
CALL JOB:SEARCH-R1-S13D
SET P045 P006
SFTON3D P045
SMOVL C00163 BC00163 V=60.0  +MOVJ EC00163
SMOVL C00164 BC00164 V=60.0  +MOVJ EC00164
SREFP 3 C00165 BC00165  +REFP EC00165
CALL JOB:SEARCH-R1-S13D
SET P045 P006
SFTON3D P045
SMOVL C00166 BC00166 V=60.0  +MOVJ EC00166
SMOVL C00167 BC00167 V=60.0  +MOVJ EC00167
SREFP 3 C00168 BC00168  +REFP EC00168
CALL JOB:SEARCH-R1-S13D
SET P045 P006
SFTON3D P045
SMOVL C00169 BC00169 V=60.0  +MOVJ EC00169
MOVL C00170 BC00170 V=400.0  +MOVJ EC00170 VJ=100.00
MOVL C00171 BC00171 V=1000.0  +MOVJ EC00171 VJ=100.00
MOVL C00172 BC00172 V=1000.0  +MOVJ EC00172 VJ=100.00
'Path S1168
SFTOF3D
MOVJ C00173 BC00173 VJ=100.00  +MOVJ EC00173 VJ=100.00
MOVL C00174 BC00174 V=400.0  +MOVJ EC00174 VJ=100.00
SMOVL C00175 BC00175 V=60.0  +MOVJ EC00175
SREFP 3 C00176 BC00176  +REFP EC00176
CALL JOB:SEARCH-R1-S13D
SET P044 P006
SFTON3D P044
SMOVL C00177 BC00177 V=60.0  +MOVJ EC00177
SMOVL C00178 BC00178 V=60.0  +MOVJ EC00178
SREFP 3 C00179 BC00179  +REFP EC00179
CALL JOB:SEARCH-R1-S13D
SET P044 P006
SFTON3D P044
SMOVL C00180 BC00180 V=60.0  +MOVJ EC00180
MOVL C00181 BC00181 V=400.0  +MOVJ EC00181 VJ=100.00
MOVL C00182 BC00182 V=1000.0  +MOVJ EC00182 VJ=100.00
'Path S1167
SFTOF3D
MOVJ C00183 BC00183 VJ=100.00  +MOVJ EC00183 VJ=100.00
MOVL C00184 BC00184 V=400.0  +MOVJ EC00184 VJ=100.00
SMOVL C00185 BC00185 V=60.0  +MOVJ EC00185
SREFP 3 C00186 BC00186  +REFP EC00186
CALL JOB:SEARCH-R1-S13D
SET P043 P006
SFTON3D P043
SMOVL C00187 BC00187 V=60.0  +MOVJ EC00187
SMOVL C00188 BC00188 V=60.0  +MOVJ EC00188
SREFP 3 C00189 BC00189  +REFP EC00189
CALL JOB:SEARCH-R1-S13D
SET P043 P006
SFTON3D P043
SMOVL C00190 BC00190 V=60.0  +MOVJ EC00190
SMOVL C00191 BC00191 V=60.0  +MOVJ EC00191
SREFP 3 C00192 BC00192  +REFP EC00192
CALL JOB:SEARCH-R1-S13D
SET P043 P006
SFTON3D P043
SMOVL C00193 BC00193 V=60.0  +MOVJ EC00193
MOVL C00194 BC00194 V=400.0  +MOVJ EC00194 VJ=100.00
MOVL C00195 BC00195 V=1000.0  +MOVJ EC00195 VJ=100.00
'Path S1166
SFTOF3D
MOVJ C00196 BC00196 VJ=100.00  +MOVJ EC00196 VJ=100.00
MOVL C00197 BC00197 V=400.0  +MOVJ EC00197 VJ=100.00
SMOVL C00198 BC00198 V=60.0  +MOVJ EC00198
SREFP 3 C00199 BC00199  +REFP EC00199
CALL JOB:SEARCH-R1-S13D
SET P042 P006
SFTON3D P042
SMOVL C00200 BC00200 V=60.0  +MOVJ EC00200
SMOVL C00201 BC00201 V=60.0  +MOVJ EC00201
SREFP 3 C00202 BC00202  +REFP EC00202
CALL JOB:SEARCH-R1-S13D
SET P042 P006
SFTON3D P042
SMOVL C00203 BC00203 V=60.0  +MOVJ EC00203
SMOVL C00204 BC00204 V=60.0  +MOVJ EC00204
SREFP 3 C00205 BC00205  +REFP EC00205
CALL JOB:SEARCH-R1-S13D
SET P042 P006
SFTON3D P042
SMOVL C00206 BC00206 V=60.0  +MOVJ EC00206
MOVL C00207 BC00207 V=400.0  +MOVJ EC00207 VJ=100.00
MOVL C00208 BC00208 V=1000.0  +MOVJ EC00208 VJ=100.00
'Path S1165
SFTOF3D
MOVJ C00209 BC00209 VJ=100.00  +MOVJ EC00209 VJ=100.00
MOVL C00210 BC00210 V=400.0  +MOVJ EC00210 VJ=100.00
SMOVL C00211 BC00211 V=60.0  +MOVJ EC00211
SREFP 3 C00212 BC00212  +REFP EC00212
CALL JOB:SEARCH-R1-S13D
SET P041 P006
SFTON3D P041
SMOVL C00213 BC00213 V=60.0  +MOVJ EC00213
SMOVL C00214 BC00214 V=60.0  +MOVJ EC00214
SREFP 3 C00215 BC00215  +REFP EC00215
CALL JOB:SEARCH-R1-S13D
SET P041 P006
SFTON3D P041
SMOVL C00216 BC00216 V=60.0  +MOVJ EC00216
SMOVL C00217 BC00217 V=60.0  +MOVJ EC00217
SREFP 3 C00218 BC00218  +REFP EC00218
CALL JOB:SEARCH-R1-S13D
SET P041 P006
SFTON3D P041
SMOVL C00219 BC00219 V=60.0  +MOVJ EC00219
MOVL C00220 BC00220 V=400.0  +MOVJ EC00220 VJ=100.00
MOVL C00221 BC00221 V=1000.0  +MOVJ EC00221 VJ=100.00
'Path W378
SFTOF3D
SFTON3D P041
MOVJ C00222 BC00222 VJ=100.00  +MOVJ EC00222 VJ=100.00
SMOVL C00223 BC00223 V=400.0  +MOVJ EC00223
SMOVL C00224 BC00224 V=100.0 PL=0  +MOVJ EC00224
SREFP 1 C00225 BC00225  +REFP EC00225
SREFP 2 C00226 BC00226  +REFP EC00226
MACRO1 MJ#(0) ARGF0
ARCON
SMOVL C00227 BC00227 V=10.0  +MOVJ EC00227
SMOVL C00228 BC00228 V=10.0  +MOVJ EC00228
SMOVL C00229 BC00229 V=10.0  +MOVJ EC00229
ARCOF
SMOVL C00230 BC00230 V=400.0  +MOVJ EC00230
SMOVL C00231 BC00231 V=1000.0  +MOVJ EC00231
SFTOF3D
'Path W379
SFTOF3D
SFTON3D P042
MOVJ C00232 BC00232 VJ=100.00  +MOVJ EC00232 VJ=100.00
MOVJ C00233 BC00233 VJ=100.00  +MOVJ EC00233 VJ=100.00
SMOVL C00234 BC00234 V=400.0  +MOVJ EC00234
SMOVL C00235 BC00235 V=100.0 PL=0  +MOVJ EC00235
SREFP 1 C00236 BC00236  +REFP EC00236
SREFP 2 C00237 BC00237  +REFP EC00237
MACRO1 MJ#(0) ARGF0
ARCON
SMOVL C00238 BC00238 V=10.0  +MOVJ EC00238
SMOVL C00239 BC00239 V=10.0  +MOVJ EC00239
SMOVL C00240 BC00240 V=10.0  +MOVJ EC00240
ARCOF
SMOVL C00241 BC00241 V=400.0  +MOVJ EC00241
SMOVL C00242 BC00242 V=1000.0  +MOVJ EC00242
SFTOF3D
MOVJ C00243 BC00243 VJ=100.00  +MOVJ EC00243 VJ=100.00
'Path W380
SFTOF3D
SFTON3D P043
MOVJ C00244 BC00244 VJ=100.00  +MOVJ EC00244 VJ=100.00
MOVJ C00245 BC00245 VJ=100.00  +MOVJ EC00245 VJ=100.00
SMOVL C00246 BC00246 V=400.0  +MOVJ EC00246
SMOVL C00247 BC00247 V=100.0 PL=0  +MOVJ EC00247
SREFP 1 C00248 BC00248  +REFP EC00248
SREFP 2 C00249 BC00249  +REFP EC00249
MACRO1 MJ#(0) ARGF0
ARCON
SMOVL C00250 BC00250 V=10.0  +MOVJ EC00250
SMOVL C00251 BC00251 V=10.0  +MOVJ EC00251
SMOVL C00252 BC00252 V=10.0  +MOVJ EC00252
ARCOF
SMOVL C00253 BC00253 V=400.0  +MOVJ EC00253
SMOVL C00254 BC00254 V=1000.0  +MOVJ EC00254
SMOVL C00255 BC00255 V=1000.0  +MOVJ EC00255
SFTOF3D
'Path W381
SFTOF3D
SFTON3D P044
MOVJ C00256 BC00256 VJ=100.00  +MOVJ EC00256 VJ=100.00
SMOVL C00257 BC00257 V=400.0  +MOVJ EC00257
SMOVL C00258 BC00258 V=100.0 PL=0  +MOVJ EC00258
SREFP 1 C00259 BC00259  +REFP EC00259
SREFP 2 C00260 BC00260  +REFP EC00260
MACRO1 MJ#(0) ARGF0
ARCON
SMOVL C00261 BC00261 V=10.0  +MOVJ EC00261
SMOVL C00262 BC00262 V=10.0  +MOVJ EC00262
SMOVL C00263 BC00263 V=10.0  +MOVJ EC00263
SMOVL C00264 BC00264 V=10.0  +MOVJ EC00264
SMOVL C00265 BC00265 V=10.0  +MOVJ EC00265
SMOVL C00266 BC00266 V=10.0  +MOVJ EC00266
SMOVL C00267 BC00267 V=10.0  +MOVJ EC00267
SMOVL C00268 BC00268 V=10.0  +MOVJ EC00268
SMOVL C00269 BC00269 V=10.0  +MOVJ EC00269
SMOVL C00270 BC00270 V=10.0  +MOVJ EC00270
SMOVL C00271 BC00271 V=10.0  +MOVJ EC00271
SMOVL C00272 BC00272 V=10.0  +MOVJ EC00272
SMOVL C00273 BC00273 V=10.0  +MOVJ EC00273
SMOVL C00274 BC00274 V=10.0  +MOVJ EC00274
SMOVL C00275 BC00275 V=10.0  +MOVJ EC00275
SMOVL C00276 BC00276 V=10.0  +MOVJ EC00276
SMOVL C00277 BC00277 V=10.0  +MOVJ EC00277
SMOVL C00278 BC00278 V=10.0  +MOVJ EC00278
SMOVL C00279 BC00279 V=10.0  +MOVJ EC00279
SMOVL C00280 BC00280 V=10.0  +MOVJ EC00280
SMOVL C00281 BC00281 V=10.0  +MOVJ EC00281
SMOVL C00282 BC00282 V=10.0  +MOVJ EC00282
SMOVL C00283 BC00283 V=10.0  +MOVJ EC00283
SMOVL C00284 BC00284 V=10.0  +MOVJ EC00284
SMOVL C00285 BC00285 V=10.0  +MOVJ EC00285
ARCOF
SMOVL C00286 BC00286 V=400.0  +MOVJ EC00286
SMOVL C00287 BC00287 V=1000.0  +MOVJ EC00287
SFTOF3D
'Path W382
SFTOF3D
SFTON3D P045
MOVJ C00288 BC00288 VJ=100.00  +MOVJ EC00288 VJ=100.00
SMOVL C00289 BC00289 V=400.0  +MOVJ EC00289
SMOVL C00290 BC00290 V=100.0 PL=0  +MOVJ EC00290
SREFP 1 C00291 BC00291  +REFP EC00291
SREFP 2 C00292 BC00292  +REFP EC00292
MACRO1 MJ#(0) ARGF0
ARCON
SMOVL C00293 BC00293 V=10.0  +MOVJ EC00293
SMOVL C00294 BC00294 V=10.0  +MOVJ EC00294
SMOVL C00295 BC00295 V=10.0  +MOVJ EC00295
ARCOF
SMOVL C00296 BC00296 V=400.0  +MOVJ EC00296
SMOVL C00297 BC00297 V=1000.0  +MOVJ EC00297
SMOVL C00298 BC00298 V=1000.0  +MOVJ EC00298
SFTOF3D
MOVJ C00299 BC00299 VJ=100.00  +MOVJ EC00299 VJ=100.00
'Path W383
SFTOF3D
SFTON3D P046
MOVJ C00300 BC00300 VJ=100.00  +MOVJ EC00300 VJ=100.00
MOVJ C00301 BC00301 VJ=100.00  +MOVJ EC00301 VJ=100.00
SMOVL C00302 BC00302 V=400.0  +MOVJ EC00302
SMOVL C00303 BC00303 V=100.0 PL=0  +MOVJ EC00303
SREFP 1 C00304 BC00304  +REFP EC00304
SREFP 2 C00305 BC00305  +REFP EC00305
MACRO1 MJ#(0) ARGF0
ARCON
SMOVL C00306 BC00306 V=10.0  +MOVJ EC00306
SMOVL C00307 BC00307 V=10.0  +MOVJ EC00307
SMOVL C00308 BC00308 V=10.0  +MOVJ EC00308
ARCOF
SMOVL C00309 BC00309 V=400.0  +MOVJ EC00309
SMOVL C00310 BC00310 V=1000.0  +MOVJ EC00310
SFTOF3D
MOVJ C00311 BC00311 VJ=100.00  +MOVJ EC00311 VJ=100.00
MOVJ C00312 BC00312 VJ=100.00  +MOVJ EC00312 VJ=100.00
'Down
MOVJ C00313 BC00313 VJ=100.00  +MOVJ EC00313 VJ=100.00
MOVJ C00314 BC00314 VJ=100.00  +MOVJ EC00314 VJ=100.00
'Path W1720
SFTOF3D
SFTON3D P032
MOVJ C00315 BC00315 VJ=100.00  +MOVJ EC00315 VJ=100.00
SMOVL C00316 BC00316 V=400.0  +MOVJ EC00316
SMOVL C00317 BC00317 V=100.0 PL=0  +MOVJ EC00317
SREFP 1 C00318 BC00318  +REFP EC00318
SREFP 2 C00319 BC00319  +REFP EC00319
MACRO1 MJ#(0) ARGF0
ARCON
SMOVL C00320 BC00320 V=10.0  +MOVJ EC00320
SMOVL C00321 BC00321 V=10.0  +MOVJ EC00321
SMOVL C00322 BC00322 V=10.0  +MOVJ EC00322
SMOVL C00323 BC00323 V=10.0  +MOVJ EC00323
SMOVL C00324 BC00324 V=10.0  +MOVJ EC00324
SMOVL C00325 BC00325 V=10.0  +MOVJ EC00325
SMOVL C00326 BC00326 V=10.0  +MOVJ EC00326
SMOVL C00327 BC00327 V=10.0  +MOVJ EC00327
SMOVL C00328 BC00328 V=10.0  +MOVJ EC00328
SMOVL C00329 BC00329 V=10.0  +MOVJ EC00329
SMOVL C00330 BC00330 V=10.0  +MOVJ EC00330
SMOVL C00331 BC00331 V=10.0  +MOVJ EC00331
SMOVL C00332 BC00332 V=10.0  +MOVJ EC00332
SMOVL C00333 BC00333 V=10.0  +MOVJ EC00333
SMOVL C00334 BC00334 V=10.0  +MOVJ EC00334
ARCOF
SMOVL C00335 BC00335 V=400.0  +MOVJ EC00335
SMOVL C00336 BC00336 V=1000.0  +MOVJ EC00336
SFTOF3D
MOVJ C00337 BC00337 VJ=100.00  +MOVJ EC00337 VJ=100.00
MOVJ C00338 BC00338 VJ=100.00  +MOVJ EC00338 VJ=100.00
MOVJ C00339 BC00339 VJ=100.00  +MOVJ EC00339 VJ=100.00
MOVJ C00340 BC00340 VJ=100.00  +MOVJ EC00340 VJ=100.00
MOVJ C00341 BC00341 VJ=100.00  +MOVJ EC00341 VJ=100.00
'Path W1626
SFTOF3D
SFTON3D P022
MOVJ C00342 BC00342 VJ=100.00  +MOVJ EC00342 VJ=100.00
SMOVL C00343 BC00343 V=100.0  +MOVJ EC00343
SMOVL C00344 BC00344 V=100.0 PL=0  +MOVJ EC00344
SREFP 1 C00345 BC00345  +REFP EC00345
SREFP 2 C00346 BC00346  +REFP EC00346
MACRO1 MJ#(0) ARGF0
ARCON
SMOVL C00347 BC00347 V=10.0  +MOVJ EC00347
SMOVL C00348 BC00348 V=10.0  +MOVJ EC00348
SMOVL C00349 BC00349 V=10.0  +MOVJ EC00349
SMOVL C00350 BC00350 V=10.0  +MOVJ EC00350
SMOVL C00351 BC00351 V=10.0  +MOVJ EC00351
SMOVL C00352 BC00352 V=10.0  +MOVJ EC00352
SMOVL C00353 BC00353 V=10.0  +MOVJ EC00353
ARCOF
SMOVL C00354 BC00354 V=400.0  +MOVJ EC00354
SMOVL C00355 BC00355 V=1000.0  +MOVJ EC00355
SFTOF3D
'Path W1627
SFTOF3D
SFTON3D P022
MOVJ C00356 BC00356 VJ=100.00  +MOVJ EC00356 VJ=100.00
SMOVL C00357 BC00357 V=100.0  +MOVJ EC00357
SMOVL C00358 BC00358 V=100.0 PL=0  +MOVJ EC00358
SREFP 1 C00359 BC00359  +REFP EC00359
SREFP 2 C00360 BC00360  +REFP EC00360
MACRO1 MJ#(0) ARGF0
ARCON
SMOVL C00361 BC00361 V=10.0  +MOVJ EC00361
SMOVL C00362 BC00362 V=10.0  +MOVJ EC00362
SMOVL C00363 BC00363 V=10.0  +MOVJ EC00363
ARCOF
SMOVL C00364 BC00364 V=400.0  +MOVJ EC00364
SMOVL C00365 BC00365 V=1000.0  +MOVJ EC00365
SFTOF3D
MOVJ C00366 BC00366 VJ=100.00  +MOVJ EC00366 VJ=100.00
'
'Path W1629
SFTOF3D
SFTON3D P023
MOVJ C00367 BC00367 VJ=100.00  +MOVJ EC00367 VJ=100.00
MOVJ C00368 BC00368 VJ=100.00  +MOVJ EC00368 VJ=100.00
SMOVL C00369 BC00369 V=400.0  +MOVJ EC00369
SMOVL C00370 BC00370 V=100.0 PL=0  +MOVJ EC00370
SREFP 1 C00371 BC00371  +REFP EC00371
SREFP 2 C00372 BC00372  +REFP EC00372
MACRO1 MJ#(0) ARGF0
ARCON
SMOVL C00373 BC00373 V=10.0  +MOVJ EC00373
SMOVL C00374 BC00374 V=10.0  +MOVJ EC00374
SMOVL C00375 BC00375 V=10.0  +MOVJ EC00375
ARCOF
SMOVL C00376 BC00376 V=400.0  +MOVJ EC00376
SMOVL C00377 BC00377 V=1000.0  +MOVJ EC00377
SFTOF3D
'Path W1630
SFTOF3D
SFTON3D P023
MOVJ C00378 BC00378 VJ=100.00  +MOVJ EC00378 VJ=100.00
SMOVL C00379 BC00379 V=100.0  +MOVJ EC00379
SMOVL C00380 BC00380 V=100.0 PL=0  +MOVJ EC00380
SREFP 1 C00381 BC00381  +REFP EC00381
SREFP 2 C00382 BC00382  +REFP EC00382
MACRO1 MJ#(0) ARGF0
ARCON
SMOVL C00383 BC00383 V=10.0  +MOVJ EC00383
SMOVL C00384 BC00384 V=10.0  +MOVJ EC00384
SMOVL C00385 BC00385 V=10.0  +MOVJ EC00385
ARCOF
SMOVL C00386 BC00386 V=400.0  +MOVJ EC00386
SMOVL C00387 BC00387 V=1000.0  +MOVJ EC00387
SMOVL C00388 BC00388 V=1000.0  +MOVJ EC00388
SFTOF3D
'Path W1631
SFTOF3D
SFTON3D P023
MOVJ C00389 BC00389 VJ=100.00  +MOVJ EC00389 VJ=100.00
SMOVL C00390 BC00390 V=100.0  +MOVJ EC00390
SMOVL C00391 BC00391 V=100.0 PL=0  +MOVJ EC00391
SREFP 1 C00392 BC00392  +REFP EC00392
SREFP 2 C00393 BC00393  +REFP EC00393
MACRO1 MJ#(0) ARGF0
ARCON
SMOVL C00394 BC00394 V=10.0  +MOVJ EC00394
ARCOF
SMOVL C00395 BC00395 V=400.0  +MOVJ EC00395
SMOVL C00396 BC00396 V=1000.0  +MOVJ EC00396
SFTOF3D
'
'Path W1632
SFTOF3D
SFTON3D P024
MOVJ C00397 BC00397 VJ=100.00  +MOVJ EC00397 VJ=100.00
SMOVL C00398 BC00398 V=100.0  +MOVJ EC00398
SMOVL C00399 BC00399 V=100.0 PL=0  +MOVJ EC00399
SREFP 1 C00400 BC00400  +REFP EC00400
SREFP 2 C00401 BC00401  +REFP EC00401
MACRO1 MJ#(0) ARGF0
ARCON
SMOVL C00402 BC00402 V=10.0  +MOVJ EC00402
SMOVL C00403 BC00403 V=10.0  +MOVJ EC00403
SMOVL C00404 BC00404 V=10.0  +MOVJ EC00404
ARCOF
SMOVL C00405 BC00405 V=400.0  +MOVJ EC00405
SMOVL C00406 BC00406 V=1000.0  +MOVJ EC00406
SFTOF3D
'Path W1633
SFTOF3D
SFTON3D P024
MOVJ C00407 BC00407 VJ=100.00  +MOVJ EC00407 VJ=100.00
SMOVL C00408 BC00408 V=100.0  +MOVJ EC00408
SMOVL C00409 BC00409 V=100.0 PL=0  +MOVJ EC00409
SREFP 1 C00410 BC00410  +REFP EC00410
SREFP 2 C00411 BC00411  +REFP EC00411
MACRO1 MJ#(0) ARGF0
ARCON
SMOVL C00412 BC00412 V=10.0  +MOVJ EC00412
SMOVL C00413 BC00413 V=10.0  +MOVJ EC00413
SMOVL C00414 BC00414 V=10.0  +MOVJ EC00414
ARCOF
SMOVL C00415 BC00415 V=400.0  +MOVJ EC00415
SMOVL C00416 BC00416 V=1000.0  +MOVJ EC00416
SMOVL C00417 BC00417 V=1000.0  +MOVJ EC00417
SFTOF3D
'Path W1634
SFTOF3D
SFTON3D P024
MOVJ C00418 BC00418 VJ=100.00  +MOVJ EC00418 VJ=100.00
SMOVL C00419 BC00419 V=100.0  +MOVJ EC00419
SMOVL C00420 BC00420 V=100.0 PL=0  +MOVJ EC00420
SREFP 1 C00421 BC00421  +REFP EC00421
SREFP 2 C00422 BC00422  +REFP EC00422
MACRO1 MJ#(0) ARGF0
ARCON
SMOVL C00423 BC00423 V=10.0  +MOVJ EC00423
ARCOF
SMOVL C00424 BC00424 V=400.0  +MOVJ EC00424
SMOVL C00425 BC00425 V=1000.0  +MOVJ EC00425
SFTOF3D
'
'Path W1635
SFTOF3D
SFTON3D P025
MOVJ C00426 BC00426 VJ=100.00  +MOVJ EC00426 VJ=100.00
SMOVL C00427 BC00427 V=100.0  +MOVJ EC00427
SMOVL C00428 BC00428 V=100.0 PL=0  +MOVJ EC00428
SREFP 1 C00429 BC00429  +REFP EC00429
SREFP 2 C00430 BC00430  +REFP EC00430
MACRO1 MJ#(0) ARGF0
ARCON
SMOVL C00431 BC00431 V=10.0  +MOVJ EC00431
SMOVL C00432 BC00432 V=10.0  +MOVJ EC00432
SMOVL C00433 BC00433 V=10.0  +MOVJ EC00433
ARCOF
SMOVL C00434 BC00434 V=400.0  +MOVJ EC00434
SMOVL C00435 BC00435 V=1000.0  +MOVJ EC00435
SFTOF3D
'Path W1636
SFTOF3D
SFTON3D P025
MOVJ C00436 BC00436 VJ=100.00  +MOVJ EC00436 VJ=100.00
SMOVL C00437 BC00437 V=100.0  +MOVJ EC00437
SMOVL C00438 BC00438 V=100.0 PL=0  +MOVJ EC00438
SREFP 1 C00439 BC00439  +REFP EC00439
SREFP 2 C00440 BC00440  +REFP EC00440
MACRO1 MJ#(0) ARGF0
ARCON
SMOVL C00441 BC00441 V=10.0  +MOVJ EC00441
SMOVL C00442 BC00442 V=10.0  +MOVJ EC00442
SMOVL C00443 BC00443 V=10.0  +MOVJ EC00443
ARCOF
SMOVL C00444 BC00444 V=400.0  +MOVJ EC00444
SMOVL C00445 BC00445 V=1000.0  +MOVJ EC00445
SMOVL C00446 BC00446 V=1000.0  +MOVJ EC00446
SFTOF3D
'Path W1637
SFTOF3D
SFTON3D P025
MOVJ C00447 BC00447 VJ=100.00  +MOVJ EC00447 VJ=100.00
SMOVL C00448 BC00448 V=100.0  +MOVJ EC00448
SMOVL C00449 BC00449 V=100.0 PL=0  +MOVJ EC00449
SREFP 1 C00450 BC00450  +REFP EC00450
SREFP 2 C00451 BC00451  +REFP EC00451
MACRO1 MJ#(0) ARGF0
ARCON
SMOVL C00452 BC00452 V=10.0  +MOVJ EC00452
ARCOF
SMOVL C00453 BC00453 V=400.0  +MOVJ EC00453
SMOVL C00454 BC00454 V=1000.0  +MOVJ EC00454
SFTOF3D
MOVJ C00455 BC00455 VJ=100.00  +MOVJ EC00455 VJ=100.00
MOVJ C00456 BC00456 VJ=100.00  +MOVJ EC00456 VJ=100.00
MOVJ C00457 BC00457 VJ=100.00  +MOVJ EC00457 VJ=100.00
'
'Path W1639
SFTOF3D
SFTON3D P023
SMOVL C00458 BC00458 V=100.0  +MOVJ EC00458
SMOVL C00459 BC00459 V=100.0 PL=0  +MOVJ EC00459
SREFP 1 C00460 BC00460  +REFP EC00460
SREFP 2 C00461 BC00461  +REFP EC00461
MACRO1 MJ#(0) ARGF0
ARCON
SMOVL C00462 BC00462 V=10.0  +MOVJ EC00462
SMOVL C00463 BC00463 V=10.0  +MOVJ EC00463
SMOVL C00464 BC00464 V=10.0  +MOVJ EC00464
ARCOF
SMOVL C00465 BC00465 V=400.0  +MOVJ EC00465
SFTOF3D
'Path W1638
SFTOF3D
SFTON3D P023
SMOVL C00466 BC00466 V=100.0  +MOVJ EC00466
SMOVL C00467 BC00467 V=100.0 PL=0  +MOVJ EC00467
SREFP 1 C00468 BC00468  +REFP EC00468
SREFP 2 C00469 BC00469  +REFP EC00469
MACRO1 MJ#(0) ARGF0
ARCON
SMOVL C00470 BC00470 V=10.0  +MOVJ EC00470
SMOVL C00471 BC00471 V=10.0  +MOVJ EC00471
SMOVL C00472 BC00472 V=10.0  +MOVJ EC00472
ARCOF
SMOVL C00473 BC00473 V=400.0  +MOVJ EC00473
SFTOF3D
MOVJ C00474 BC00474 VJ=100.00  +MOVJ EC00474 VJ=100.00
'
'Path W1640
SFTOF3D
SFTON3D P024
MOVJ C00475 BC00475 VJ=100.00  +MOVJ EC00475 VJ=100.00
MOVJ C00476 BC00476 VJ=100.00  +MOVJ EC00476 VJ=100.00
SMOVL C00477 BC00477 V=400.0  +MOVJ EC00477
SMOVL C00478 BC00478 V=100.0 PL=0  +MOVJ EC00478
SREFP 1 C00479 BC00479  +REFP EC00479
SREFP 2 C00480 BC00480  +REFP EC00480
MACRO1 MJ#(0) ARGF0
ARCON
SMOVL C00481 BC00481 V=10.0  +MOVJ EC00481
SMOVL C00482 BC00482 V=10.0  +MOVJ EC00482
SMOVL C00483 BC00483 V=10.0  +MOVJ EC00483
ARCOF
SMOVL C00484 BC00484 V=400.0  +MOVJ EC00484
SMOVL C00485 BC00485 V=1000.0  +MOVJ EC00485
SMOVL C00486 BC00486 V=1000.0  +MOVJ EC00486
SFTOF3D
'Path W1641
SFTOF3D
SFTON3D P025
SMOVL C00487 BC00487 V=100.0  +MOVJ EC00487
SMOVL C00488 BC00488 V=100.0 PL=0  +MOVJ EC00488
SREFP 1 C00489 BC00489  +REFP EC00489
SREFP 2 C00490 BC00490  +REFP EC00490
MACRO1 MJ#(0) ARGF0
ARCON
SMOVL C00491 BC00491 V=10.0  +MOVJ EC00491
SMOVL C00492 BC00492 V=10.0  +MOVJ EC00492
SMOVL C00493 BC00493 V=10.0  +MOVJ EC00493
ARCOF
SMOVL C00494 BC00494 V=400.0  +MOVJ EC00494
SMOVL C00495 BC00495 V=1000.0  +MOVJ EC00495
SMOVL C00496 BC00496 V=1000.0  +MOVJ EC00496
SFTOF3D
MOVJ C00497 BC00497 VJ=100.00  +MOVJ EC00497 VJ=100.00
MOVJ C00498 BC00498 VJ=100.00  +MOVJ EC00498 VJ=100.00
MOVJ C00499 BC00499 VJ=100.00  +MOVJ EC00499 VJ=100.00
MOVJ C00500 BC00500 VJ=100.00  +MOVJ EC00500 VJ=100.00
'Path W1911
SFTOF3D
SFTON3D P021
MOVJ C00501 BC00501 VJ=100.00  +MOVJ EC00501 VJ=100.00
SMOVL C00502 BC00502 V=100.0  +MOVJ EC00502
SMOVL C00503 BC00503 V=100.0 PL=0  +MOVJ EC00503
SREFP 1 C00504 BC00504  +REFP EC00504
SREFP 2 C00505 BC00505  +REFP EC00505
MACRO1 MJ#(0) ARGF0
ARCON
SMOVL C00506 BC00506 V=10.0  +MOVJ EC00506
SMOVL C00507 BC00507 V=10.0  +MOVJ EC00507
SMOVL C00508 BC00508 V=10.0  +MOVJ EC00508
SMOVL C00509 BC00509 V=10.0  +MOVJ EC00509
SMOVL C00510 BC00510 V=10.0  +MOVJ EC00510
SMOVL C00511 BC00511 V=10.0  +MOVJ EC00511
SMOVL C00512 BC00512 V=10.0  +MOVJ EC00512
SMOVL C00513 BC00513 V=10.0  +MOVJ EC00513
SMOVL C00514 BC00514 V=10.0  +MOVJ EC00514
SMOVL C00515 BC00515 V=10.0  +MOVJ EC00515
ARCOF
SMOVL C00516 BC00516 V=400.0  +MOVJ EC00516
SMOVL C00517 BC00517 V=1000.0  +MOVJ EC00517
SFTOF3D
MOVJ C00518 BC00518 VJ=100.00  +MOVJ EC00518 VJ=100.00
MOVJ C00519 BC00519 VJ=100.00  +MOVJ EC00519 VJ=100.00
'
MOVJ C00520 BC00520 VJ=100.00  +MOVJ EC00520 VJ=100.00
MOVJ C00521 BC00521 VJ=100.00  +MOVJ EC00521 VJ=100.00
'Path W1642
SFTOF3D
SFTON3D P024
MOVJ C00522 BC00522 VJ=100.00  +MOVJ EC00522 VJ=100.00
SMOVL C00523 BC00523 V=100.0  +MOVJ EC00523
SMOVL C00524 BC00524 V=100.0 PL=0  +MOVJ EC00524
SREFP 1 C00525 BC00525  +REFP EC00525
SREFP 2 C00526 BC00526  +REFP EC00526
MACRO1 MJ#(0) ARGF0
ARCON
SMOVL C00527 BC00527 V=10.0  +MOVJ EC00527
SMOVL C00528 BC00528 V=10.0  +MOVJ EC00528
SMOVL C00529 BC00529 V=10.0  +MOVJ EC00529
ARCOF
SMOVL C00530 BC00530 V=400.0  +MOVJ EC00530
SMOVL C00531 BC00531 V=1000.0  +MOVJ EC00531
SFTOF3D
'Path W1643
SFTOF3D
SFTON3D P025
MOVJ C00532 BC00532 VJ=100.00  +MOVJ EC00532 VJ=100.00
SMOVL C00533 BC00533 V=100.0  +MOVJ EC00533
SMOVL C00534 BC00534 V=100.0 PL=0  +MOVJ EC00534
SREFP 1 C00535 BC00535  +REFP EC00535
SREFP 2 C00536 BC00536  +REFP EC00536
MACRO1 MJ#(0) ARGF0
ARCON
SMOVL C00537 BC00537 V=10.0  +MOVJ EC00537
SMOVL C00538 BC00538 V=10.0  +MOVJ EC00538
SMOVL C00539 BC00539 V=10.0  +MOVJ EC00539
ARCOF
SMOVL C00540 BC00540 V=400.0  +MOVJ EC00540
SMOVL C00541 BC00541 V=1000.0  +MOVJ EC00541
SMOVL C00542 BC00542 V=1000.0  +MOVJ EC00542
SFTOF3D
'
'Path W1644
SFTOF3D
SFTON3D P026
MOVJ C00543 BC00543 VJ=100.00  +MOVJ EC00543 VJ=100.00
SMOVL C00544 BC00544 V=100.0  +MOVJ EC00544
SMOVL C00545 BC00545 V=100.0 PL=0  +MOVJ EC00545
SREFP 1 C00546 BC00546  +REFP EC00546
SREFP 2 C00547 BC00547  +REFP EC00547
MACRO1 MJ#(0) ARGF0
ARCON
SMOVL C00548 BC00548 V=10.0  +MOVJ EC00548
SMOVL C00549 BC00549 V=10.0  +MOVJ EC00549
SMOVL C00550 BC00550 V=10.0  +MOVJ EC00550
ARCOF
SMOVL C00551 BC00551 V=400.0  +MOVJ EC00551
SMOVL C00552 BC00552 V=1000.0  +MOVJ EC00552
SFTOF3D
'Path W1645
SFTOF3D
SFTON3D P027
MOVJ C00553 BC00553 VJ=100.00  +MOVJ EC00553 VJ=100.00
SMOVL C00554 BC00554 V=100.0  +MOVJ EC00554
SMOVL C00555 BC00555 V=100.0 PL=0  +MOVJ EC00555
SREFP 1 C00556 BC00556  +REFP EC00556
SREFP 2 C00557 BC00557  +REFP EC00557
MACRO1 MJ#(0) ARGF0
ARCON
SMOVL C00558 BC00558 V=10.0  +MOVJ EC00558
SMOVL C00559 BC00559 V=10.0  +MOVJ EC00559
SMOVL C00560 BC00560 V=10.0  +MOVJ EC00560
ARCOF
SMOVL C00561 BC00561 V=400.0  +MOVJ EC00561
SMOVL C00562 BC00562 V=1000.0  +MOVJ EC00562
SFTOF3D
MOVJ C00563 BC00563 VJ=100.00  +MOVJ EC00563 VJ=100.00
MOVJ C00564 BC00564 VJ=100.00  +MOVJ EC00564 VJ=100.00
'jakie searche do takicj spoin?
MOVJ C00565 BC00565 VJ=100.00  +MOVJ EC00565 VJ=100.00
'Path W1646
SFTOF3D
MOVJ C00566 BC00566 VJ=100.00  +MOVJ EC00566 VJ=100.00
MOVL C00567 BC00567 V=100.0  +MOVJ EC00567 VJ=100.00
SMOVL C00568 BC00568 V=100.0 PL=0  +MOVJ EC00568
SREFP 1 C00569 BC00569  +REFP EC00569
SREFP 2 C00570 BC00570  +REFP EC00570
MACRO1 MJ#(0) ARGF0
ARCON
SMOVL C00571 BC00571 V=10.0  +MOVJ EC00571
ARCOF
MOVL C00572 BC00572 V=400.0  +MOVJ EC00572 VJ=100.00
MOVL C00573 BC00573 V=1000.0  +MOVJ EC00573 VJ=100.00
MOVL C00574 BC00574 V=1000.0  +MOVJ EC00574 VJ=100.00
MOVJ C00575 BC00575 VJ=100.00  +MOVJ EC00575 VJ=100.00
'brak dostÄpu do jednej spoiny
'Path W1647
SFTOF3D
MOVJ C00576 BC00576 VJ=100.00  +MOVJ EC00576 VJ=100.00
MOVJ C00577 BC00577 VJ=100.00  +MOVJ EC00577 VJ=100.00
MOVL C00578 BC00578 V=400.0  +MOVJ EC00578 VJ=100.00
SMOVL C00579 BC00579 V=100.0 PL=0  +MOVJ EC00579
SREFP 1 C00580 BC00580  +REFP EC00580
SREFP 2 C00581 BC00581  +REFP EC00581
MACRO1 MJ#(0) ARGF0
ARCON
SMOVL C00582 BC00582 V=10.0  +MOVJ EC00582
ARCOF
MOVL C00583 BC00583 V=400.0  +MOVJ EC00583 VJ=100.00
MOVL C00584 BC00584 V=1000.0  +MOVJ EC00584 VJ=100.00
'Path W1648
SFTOF3D
MOVJ C00585 BC00585 VJ=100.00  +MOVJ EC00585 VJ=100.00
MOVL C00586 BC00586 V=100.0  +MOVJ EC00586 VJ=100.00
SMOVL C00587 BC00587 V=100.0 PL=0  +MOVJ EC00587
SREFP 1 C00588 BC00588  +REFP EC00588
SREFP 2 C00589 BC00589  +REFP EC00589
MACRO1 MJ#(0) ARGF0
ARCON
SMOVL C00590 BC00590 V=10.0  +MOVJ EC00590
ARCOF
MOVL C00591 BC00591 V=400.0  +MOVJ EC00591 VJ=100.00
MOVL C00592 BC00592 V=1000.0  +MOVJ EC00592 VJ=100.00
MOVL C00593 BC00593 V=1000.0  +MOVJ EC00593 VJ=100.00
MOVJ C00594 BC00594 VJ=100.00  +MOVJ EC00594 VJ=100.00
'Path W1649
SFTOF3D
MOVJ C00595 BC00595 VJ=100.00  +MOVJ EC00595 VJ=100.00
MOVL C00596 BC00596 V=100.0  +MOVJ EC00596 VJ=100.00
SMOVL C00597 BC00597 V=100.0 PL=0  +MOVJ EC00597
SREFP 1 C00598 BC00598  +REFP EC00598
SREFP 2 C00599 BC00599  +REFP EC00599
MACRO1 MJ#(0) ARGF0
ARCON
SMOVL C00600 BC00600 V=10.0  +MOVJ EC00600
ARCOF
MOVL C00601 BC00601 V=400.0  +MOVJ EC00601 VJ=100.00
MOVL C00602 BC00602 V=1000.0  +MOVJ EC00602 VJ=100.00
'Path W1650
SFTOF3D
MOVJ C00603 BC00603 VJ=100.00  +MOVJ EC00603 VJ=100.00
MOVL C00604 BC00604 V=100.0  +MOVJ EC00604 VJ=100.00
SMOVL C00605 BC00605 V=100.0 PL=0  +MOVJ EC00605
SREFP 1 C00606 BC00606  +REFP EC00606
SREFP 2 C00607 BC00607  +REFP EC00607
MACRO1 MJ#(0) ARGF0
ARCON
SMOVL C00608 BC00608 V=10.0  +MOVJ EC00608
ARCOF
MOVL C00609 BC00609 V=400.0  +MOVJ EC00609 VJ=100.00
MOVL C00610 BC00610 V=1000.0  +MOVJ EC00610 VJ=100.00
'Path W1651
SFTOF3D
MOVJ C00611 BC00611 VJ=100.00  +MOVJ EC00611 VJ=100.00
MOVL C00612 BC00612 V=100.0  +MOVJ EC00612 VJ=100.00
SMOVL C00613 BC00613 V=100.0 PL=0  +MOVJ EC00613
SREFP 1 C00614 BC00614  +REFP EC00614
SREFP 2 C00615 BC00615  +REFP EC00615
MACRO1 MJ#(0) ARGF0
ARCON
SMOVL C00616 BC00616 V=10.0  +MOVJ EC00616
ARCOF
MOVL C00617 BC00617 V=400.0  +MOVJ EC00617 VJ=100.00
MOVL C00618 BC00618 V=1000.0  +MOVJ EC00618 VJ=100.00
'Path W1652
SFTOF3D
MOVJ C00619 BC00619 VJ=100.00  +MOVJ EC00619 VJ=100.00
MOVL C00620 BC00620 V=100.0  +MOVJ EC00620 VJ=100.00
SMOVL C00621 BC00621 V=100.0 PL=0  +MOVJ EC00621
SREFP 1 C00622 BC00622  +REFP EC00622
SREFP 2 C00623 BC00623  +REFP EC00623
MACRO1 MJ#(0) ARGF0
ARCON
SMOVL C00624 BC00624 V=10.0  +MOVJ EC00624
ARCOF
MOVL C00625 BC00625 V=400.0  +MOVJ EC00625 VJ=100.00
MOVL C00626 BC00626 V=1000.0  +MOVJ EC00626 VJ=100.00
'jakie searche do takicj spoin?
MOVJ C00627 BC00627 VJ=100.00  +MOVJ EC00627 VJ=100.00
'Path W1653
SFTOF3D
MOVJ C00628 BC00628 VJ=100.00  +MOVJ EC00628 VJ=100.00
MOVL C00629 BC00629 V=100.0  +MOVJ EC00629 VJ=100.00
SMOVL C00630 BC00630 V=100.0 PL=0  +MOVJ EC00630
SREFP 1 C00631 BC00631  +REFP EC00631
SREFP 2 C00632 BC00632  +REFP EC00632
MACRO1 MJ#(0) ARGF0
ARCON
SMOVL C00633 BC00633 V=10.0  +MOVJ EC00633
SMOVL C00634 BC00634 V=10.0  +MOVJ EC00634
SMOVL C00635 BC00635 V=10.0  +MOVJ EC00635
ARCOF
MOVL C00636 BC00636 V=400.0  +MOVJ EC00636 VJ=100.00
MOVL C00637 BC00637 V=1000.0  +MOVJ EC00637 VJ=100.00
MOVL C00638 BC00638 V=1000.0  +MOVJ EC00638 VJ=100.00
'Path W1654
SFTOF3D
MOVJ C00639 BC00639 VJ=100.00  +MOVJ EC00639 VJ=100.00
MOVL C00640 BC00640 V=100.0  +MOVJ EC00640 VJ=100.00
SMOVL C00641 BC00641 V=100.0 PL=0  +MOVJ EC00641
SREFP 1 C00642 BC00642  +REFP EC00642
SREFP 2 C00643 BC00643  +REFP EC00643
MACRO1 MJ#(0) ARGF0
ARCON
SMOVL C00644 BC00644 V=10.0  +MOVJ EC00644
SMOVL C00645 BC00645 V=10.0  +MOVJ EC00645
SMOVL C00646 BC00646 V=10.0  +MOVJ EC00646
ARCOF
MOVL C00647 BC00647 V=400.0  +MOVJ EC00647 VJ=100.00
MOVL C00648 BC00648 V=1000.0  +MOVJ EC00648 VJ=100.00
MOVL C00649 BC00649 V=1000.0  +MOVJ EC00649 VJ=100.00
MOVJ C00650 BC00650 VJ=100.00  +MOVJ EC00650 VJ=100.00
MOVJ C00651 BC00651 VJ=100.00  +MOVJ EC00651 VJ=100.00
MOVJ C00652 BC00652 VJ=100.00  +MOVJ EC00652 VJ=100.00
MOVJ C00653 BC00653 VJ=100.00  +MOVJ EC00653 VJ=100.00
'68,69
MOVJ C00654 BC00654 VJ=100.00  +MOVJ EC00654 VJ=100.00
'Path W1655
SFTOF3D
SFTON3D P030
MOVJ C00655 BC00655 VJ=100.00  +MOVJ EC00655 VJ=100.00
SMOVL C00656 BC00656 V=100.0  +MOVJ EC00656
SMOVL C00657 BC00657 V=100.0 PL=0  +MOVJ EC00657
SREFP 1 C00658 BC00658  +REFP EC00658
SREFP 2 C00659 BC00659  +REFP EC00659
MACRO1 MJ#(0) ARGF0
ARCON
SFTON3D P029
SMOVL C00660 BC00660 V=10.0  +MOVJ EC00660
SMOVL C00661 BC00661 V=10.0  +MOVJ EC00661
SFTON3D P028
SMOVL C00662 BC00662 V=10.0  +MOVJ EC00662
ARCOF
SMOVL C00663 BC00663 V=400.0  +MOVJ EC00663
SMOVL C00664 BC00664 V=1000.0  +MOVJ EC00664
SFTOF3D
MOVJ C00665 BC00665 VJ=100.00  +MOVJ EC00665 VJ=100.00
MOVJ C00666 BC00666 VJ=100.00  +MOVJ EC00666 VJ=100.00
'Path W1656
SFTOF3D
SFTON3D P031
MOVJ C00667 BC00667 VJ=100.00  +MOVJ EC00667 VJ=100.00
SMOVL C00668 BC00668 V=100.0  +MOVJ EC00668
SMOVL C00669 BC00669 V=100.0 PL=0  +MOVJ EC00669
SREFP 1 C00670 BC00670  +REFP EC00670
SREFP 2 C00671 BC00671  +REFP EC00671
MACRO1 MJ#(0) ARGF0
ARCON
SMOVL C00672 BC00672 V=10.0  +MOVJ EC00672
SMOVL C00673 BC00673 V=10.0  +MOVJ EC00673
SMOVL C00674 BC00674 V=10.0  +MOVJ EC00674
ARCOF
SMOVL C00675 BC00675 V=400.0  +MOVJ EC00675
SMOVL C00676 BC00676 V=1000.0  +MOVJ EC00676
SFTOF3D
MOVJ C00677 BC00677 VJ=100.00  +MOVJ EC00677 VJ=100.00
MOVJ C00678 BC00678 VJ=100.00  +MOVJ EC00678 VJ=100.00
